KUKA KRL program: MyProgram_235().src

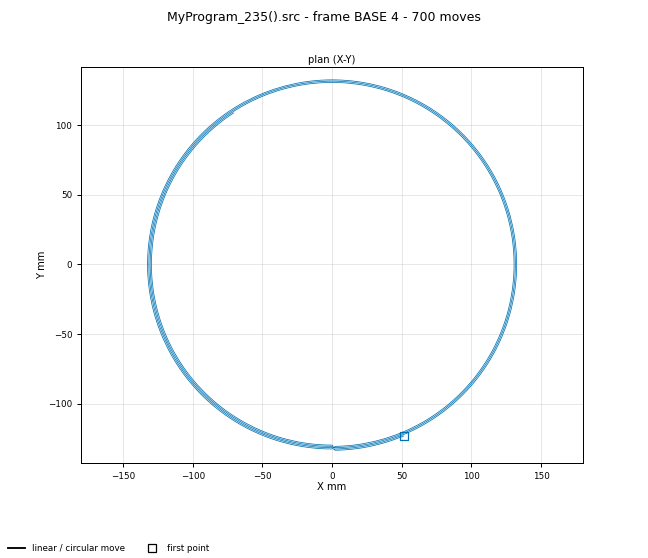
[picture p0: tool path of MyProgram_235().src in frame BASE 4, 700 of 700 moves have a stored position in this frame; points joined in program order, loops and branches not executed]
&ACCESS RVP
&REL 1
&PARAM TEMPLATE = C:\KRC\Roboter\Template\vorgabe
&PARAM EDITMASK = *
DEF MyProgram_235()
; ---- Setting reference (Base) ----
$BASE = BASE_DATA[4]

; --------------------------
; ---- Setting tool (TCP) ----
$TOOL = TOOL_DATA[3]
; --------------------------

$VEL.CP = VEL_APROX_PRINT
Startdeposition()
$VEL.CP = VEL_PRINT
LIN {X 51.31,Y -123.078,Z 159,A -69.1463,B 20.1877,C -0.5171,E1 20.2552,E2 517.2278} C_DIS
LIN {X 48.8194,Y -124.0882,Z 159,A -70.4431,B 20.1878,C -0.5093,E1 20.2518,E2 518.5433} C_DIS
LIN {X 45.4149,Y -125.3733,Z 159,A -71.9054,B 20.1878,C -0.5117,E1 20.248,E2 519.9947} C_DIS
LIN {X 42.7947,Y -126.2935,Z 159,A -73.4065,B 20.1881,C -0.497,E1 20.2439,E2 521.5347} C_DIS
LIN {X 39.7378,Y -127.2887,Z 159,A -74.6325,B 20.188,C -0.5021,E1 20.2407,E2 522.7431} C_DIS
LIN {X 36.4684,Y -128.2628,Z 159,A -75.8559,B 20.1878,C -0.511,E1 20.2375,E2 523.9381} C_DIS
LIN {X 32.9588,Y -129.208,Z 159,A -77.479,B 20.1878,C -0.5068,E1 20.2331,E2 525.5701} C_DIS
LIN {X 29.9233,Y -129.9447,Z 159,A -78.8692,B 20.1879,C -0.5035,E1 20.2293,E2 526.9673} C_DIS
LIN {X 25.1569,Y -130.9509,Z 159,A -81.0499,B 20.1881,C -0.498,E1 20.2233,E2 529.1604} C_DIS
LIN {X 20.69,Y -131.7308,Z 159,A -82.9211,B 20.1881,C -0.4999,E1 20.2181,E2 531.0236} C_DIS
LIN {X 17.7382,Y -132.161,Z 159,A -84.2195,B 20.1881,C -0.4984,E1 20.2145,E2 532.325} C_DIS
LIN {X 14.1081,Y -132.5971,Z 159,A -85.8476,B 20.1881,C -0.4951,E1 20.21,E2 533.9611} C_DIS
LIN {X 9.8352,Y -132.9824,Z 159,A -87.5814,B 20.1881,C -0.499,E1 20.2052,E2 535.6827} C_DIS
LIN {X 6.2788,Y -133.1983,Z 159,A -89.2049,B 20.1881,C -0.4945,E1 20.2006,E2 537.3184} C_DIS
LIN {X 2.1393,Y -133.3285,Z 159,A -90.8711,B 20.1881,C -0.4988,E1 20.196,E2 538.9717} C_DIS
LIN {X 2.1393,Y -133.3285,Z 159,A -90.8711,B 20.1881,C -0.4988,E1 20.196,E2 538.9717} C_DIS
Enddeposition()
LIN {X 0.915,Y -132.4111,Z 159,A -90.6799,B 18.9878,C -0.3693,E1 18.993,E2 539.0606} C_DIS
Startdeposition()
$VEL.CP = VEL_PRINT
LIN {X 3.9489,Y -132.359,Z 159,A -89.0902,B 18.9875,C -0.3807,E1 18.9975,E2 537.4365} C_DIS
LIN {X 8.1067,Y -132.1692,Z 159,A -87.3119,B 18.9875,C -0.3804,E1 19.0025,E2 535.66} C_DIS
LIN {X 11.2426,Y -131.9395,Z 159,A -85.8993,B 18.9875,C -0.3831,E1 19.0064,E2 534.2402} C_DIS
LIN {X 15.547,Y -131.5017,Z 159,A -84.0509,B 18.9875,C -0.3831,E1 19.0115,E2 532.3935} C_DIS
LIN {X 18.8161,Y -131.0738,Z 159,A -82.5998,B 18.9875,C -0.3849,E1 19.0156,E2 530.9384} C_DIS
LIN {X 23.141,Y -130.3798,Z 159,A -80.3181,B 18.9871,C -0.402,E1 19.022,E2 528.6076} C_DIS
LIN {X 27.1338,Y -129.6097,Z 159,A -79.0268,B 18.9875,C -0.3843,E1 19.0254,E2 527.3728} C_DIS
LIN {X 29.78,Y -129.0256,Z 159,A -77.8051,B 18.9875,C -0.3874,E1 19.0287,E2 526.144} C_DIS
LIN {X 33.8587,Y -128.0156,Z 159,A -75.9883,B 18.9874,C -0.389,E1 19.0336,E2 524.3258} C_DIS
LIN {X 37.1501,Y -127.0992,Z 159,A -73.7766,B 18.9867,C -0.4207,E1 19.0398,E2 522.022} C_DIS
LIN {X 42.6388,Y -125.3669,Z 159,A -72.0801,B 18.9873,C -0.3908,E1 19.0441,E2 520.4216} C_DIS
LIN {X 46.6963,Y -123.9106,Z 159,A -70.1681,B 18.9873,C -0.3951,E1 19.0491,E2 518.502} C_DIS
LIN {X 50.0421,Y -122.5986,Z 159,A -68.6914,B 18.9873,C -0.394,E1 19.0529,E2 517.0333} C_DIS
LIN {X 52.8027,Y -121.4341,Z 159,A -67.3975,B 18.9873,C -0.3957,E1 19.0562,E2 515.7384} C_DIS
LIN {X 55.6063,Y -120.1758,Z 159,A -66.0096,B 18.9872,C -0.4,E1 19.0598,E2 514.3419} C_DIS
LIN {X 59.0942,Y -118.501,Z 159,A -64.0272,B 18.9868,C -0.4154,E1 19.0648,E2 512.3197} C_DIS
LIN {X 62.2036,Y -116.8996,Z 159,A -62.8732,B 18.9871,C -0.4029,E1 19.0676,E2 511.2084} C_DIS
LIN {X 65.5736,Y -115.0431,Z 159,A -61.1039,B 18.9869,C -0.41,E1 19.0719,E2 509.4243} C_DIS
LIN {X 70.2696,Y -112.2358,Z 159,A -58.4917,B 18.9866,C -0.4245,E1 19.0782,E2 506.779} C_DIS
LIN {X 73.2793,Y -110.2952,Z 159,A -57.3437,B 18.9869,C -0.4106,E1 19.0808,E2 505.6786} C_DIS
LIN {X 76.3906,Y -108.1633,Z 159,A -55.3096,B 18.9865,C -0.4306,E1 19.0855,E2 503.5928} C_DIS
LIN {X 79.3344,Y -106.0234,Z 159,A -54.2415,B 18.9869,C -0.4125,E1 19.0878,E2 502.5853} C_DIS
LIN {X 82.0871,Y -103.9069,Z 159,A -52.6363,B 18.9867,C -0.4199,E1 19.0914,E2 500.9656} C_DIS
LIN {X 84.9344,Y -101.5923,Z 159,A -50.4502,B 18.9861,C -0.4485,E1 19.0962,E2 498.7032} C_DIS
LIN {X 88.5384,Y -98.4673,Z 159,A -48.5996,B 18.9862,C -0.4441,E1 19.1,E2 496.8764} C_DIS
LIN {X 91.2721,Y -95.9391,Z 159,A -47.5951,B 18.9867,C -0.4221,E1 19.1019,E2 495.9445} C_DIS
LIN {X 94.6689,Y -92.5885,Z 159,A -44.8289,B 18.9859,C -0.4566,E1 19.1076,E2 493.0888} C_DIS
LIN {X 97.6523,Y -89.4365,Z 159,A -42.7552,B 18.9856,C -0.4695,E1 19.1115,E2 490.988} C_DIS
LIN {X 101.2378,Y -85.357,Z 159,A -41.1575,B 18.9862,C -0.4433,E1 19.1142,E2 489.4802} C_DIS
LIN {X 104.3228,Y -81.557,Z 159,A -38.8266,B 18.9859,C -0.4578,E1 19.1183,E2 487.1199} C_DIS
LIN {X 106.4737,Y -78.7289,Z 159,A -36.881,B 18.9854,C -0.4792,E1 19.1217,E2 485.1214} C_DIS
LIN {X 109.3425,Y -74.6934,Z 159,A -35.5347,B 18.9861,C -0.451,E1 19.1237,E2 483.8704} C_DIS
LIN {X 111.0638,Y -72.1085,Z 159,A -33.9343,B 18.9857,C -0.4655,E1 19.1262,E2 482.2364} C_DIS
LIN {X 113.1829,Y -68.735,Z 159,A -32.2214,B 18.9857,C -0.4698,E1 19.1287,E2 480.5223} C_DIS
LIN {X 115.4009,Y -64.9419,Z 159,A -30.372,B 18.9855,C -0.4729,E1 19.1312,E2 478.6764} C_DIS
LIN {X 117.3378,Y -61.369,Z 159,A -28.6996,B 18.9855,C -0.4742,E1 19.1334,E2 477.0117} C_DIS
LIN {X 119.1222,Y -57.8349,Z 159,A -27.0067,B 18.9855,C -0.4783,E1 19.1355,E2 475.3187} C_DIS
LIN {X 120.4094,Y -55.1012,Z 159,A -25.6347,B 18.9852,C -0.4848,E1 19.1371,E2 473.9368} C_DIS
LIN {X 121.9652,Y -51.5668,Z 159,A -24.0045,B 18.9852,C -0.488,E1 19.1389,E2 472.309} C_DIS
LIN {X 124.4421,Y -45.2616,Z 159,A -21.3203,B 18.9852,C -0.4861,E1 19.1416,E2 469.6506} C_DIS
LIN {X 125.713,Y -41.6006,Z 159,A -19.4119,B 18.9848,C -0.5011,E1 19.1434,E2 467.7112} C_DIS
LIN {X 127.6951,Y -35.0529,Z 159,A -16.5806,B 18.9848,C -0.5045,E1 19.1456,E2 464.8912} C_DIS
LIN {X 128.3642,Y -32.5112,Z 159,A -15.4138,B 18.9846,C -0.5093,E1 19.1464,E2 463.7189} C_DIS
LIN {X 129.7937,Y -26.2296,Z 159,A -12.6235,B 18.9844,C -0.518,E1 19.1481,E2 460.924} C_DIS
LIN {X 130.7421,Y -21.0106,Z 159,A -10.3225,B 18.9842,C -0.5254,E1 19.1492,E2 458.6189} C_DIS
LIN {X 131.2848,Y -17.2825,Z 159,A -8.7108,B 18.9841,C -0.5297,E1 19.1498,E2 457.0068} C_DIS
LIN {X 131.7831,Y -12.9506,Z 159,A -6.9501,B 18.9841,C -0.5302,E1 19.1503,E2 455.2588} C_DIS
LIN {X 132.0586,Y -9.744,Z 159,A -5.47,B 18.9839,C -0.5383,E1 19.1507,E2 453.7658} C_DIS
LIN {X 132.2857,Y -5.9509,Z 159,A -3.646,B 18.9835,C -0.5511,E1 19.1509,E2 451.9174} C_DIS
LIN {X 132.4155,Y -0.8768,Z 159,A -1.6644,B 18.9835,C -0.5488,E1 19.151,E2 449.9587} C_DIS
LIN {X 132.3754,Y 3.3608,Z 159,A 0.1535,B 18.9835,C -0.5538,E1 19.151,E2 448.1401} C_DIS
LIN {X 132.2469,Y 6.7219,Z 159,A 1.588,B 18.9833,C -0.5575,E1 19.1507,E2 446.7061} C_DIS
LIN {X 132.0141,Y 10.3543,Z 159,A 3.2561,B 18.9831,C -0.5663,E1 19.1504,E2 445.0244} C_DIS
LIN {X 131.6494,Y 14.2426,Z 159,A 4.8067,B 18.9831,C -0.5656,E1 19.15,E2 443.4883} C_DIS
LIN {X 131.1522,Y 18.2677,Z 159,A 6.661,B 18.9828,C -0.5753,E1 19.1493,E2 441.6194} C_DIS
LIN {X 130.5569,Y 22.1221,Z 159,A 8.2165,B 18.9828,C -0.5748,E1 19.1486,E2 440.0777} C_DIS
LIN {X 129.5781,Y 27.2807,Z 159,A 11.5557,B 18.9812,C -0.6276,E1 19.1466,E2 436.6038} C_DIS
LIN {X 127.8681,Y 34.412,Z 159,A 13.1779,B 18.983,C -0.5706,E1 19.1457,E2 435.168} C_DIS
LIN {X 125.8783,Y 41.1045,Z 159,A 16.7762,B 18.982,C -0.6038,E1 19.1427,E2 431.496} C_DIS
LIN {X 124.582,Y 44.8736,Z 159,A 18.3588,B 18.982,C -0.6028,E1 19.1412,E2 429.9286} C_DIS
LIN {X 123.3427,Y 48.1759,Z 159,A 19.8352,B 18.982,C -0.6051,E1 19.1397,E2 428.4564} C_DIS
LIN {X 122.1018,Y 51.2397,Z 159,A 21.2099,B 18.9819,C -0.6068,E1 19.1383,E2 427.0868} C_DIS
LIN {X 120.8903,Y 54.0353,Z 159,A 22.5822,B 18.9817,C -0.6127,E1 19.1367,E2 425.7064} C_DIS
LIN {X 119.4225,Y 57.2063,Z 159,A 24.123,B 18.9815,C -0.6181,E1 19.1349,E2 424.1604} C_DIS
LIN {X 117.8596,Y 60.3613,Z 159,A 25.6041,B 18.9815,C -0.6205,E1 19.133,E2 422.6828} C_DIS
LIN {X 115.9936,Y 63.8779,Z 159,A 27.3655,B 18.9812,C -0.6267,E1 19.1307,E2 420.9149} C_DIS
LIN {X 113.9778,Y 67.4093,Z 159,A 29.1303,B 18.9811,C -0.6315,E1 19.1282,E2 419.1476} C_DIS
LIN {X 111.7699,Y 71.0102,Z 159,A 30.9547,B 18.9809,C -0.6361,E1 19.1255,E2 417.3219} C_DIS
LIN {X 109.3756,Y 74.6451,Z 159,A 32.839,B 18.9808,C -0.6409,E1 19.1226,E2 415.4356} C_DIS
LIN {X 106.7983,Y 78.2876,Z 159,A 34.7322,B 18.9807,C -0.644,E1 19.1195,E2 413.5452} C_DIS
LIN {X 104.0816,Y 81.8647,Z 159,A 36.6347,B 18.9806,C -0.6469,E1 19.1162,E2 411.6459} C_DIS
LIN {X 101.2742,Y 85.3136,Z 159,A 38.5288,B 18.9805,C -0.6501,E1 19.1129,E2 409.7539} C_DIS
LIN {X 98.4189,Y 88.5925,Z 159,A 40.6781,B 18.98,C -0.6655,E1 19.1088,E2 407.5706} C_DIS
LIN {X 96.1324,Y 91.0683,Z 159,A 41.8429,B 18.9803,C -0.6565,E1 19.1066,E2 406.4404} C_DIS
LIN {X 93.2493,Y 94.018,Z 159,A 43.6666,B 18.9801,C -0.6618,E1 19.103,E2 404.6107} C_DIS
LIN {X 90.0676,Y 97.0705,Z 159,A 45.5495,B 18.9801,C -0.6647,E1 19.0992,E2 402.7295} C_DIS
LIN {X 86.7928,Y 100.0097,Z 159,A 47.4911,B 18.9798,C -0.67,E1 19.0951,E2 400.7823} C_DIS
LIN {X 83.3209,Y 102.9199,Z 159,A 49.7722,B 18.9792,C -0.6869,E1 19.0901,E2 398.4612} C_DIS
LIN {X 80.1132,Y 105.4365,Z 159,A 50.9917,B 18.9799,C -0.6676,E1 19.0876,E2 397.3067} C_DIS
LIN {X 77.3722,Y 107.4641,Z 159,A 52.6714,B 18.9795,C -0.6785,E1 19.0837,E2 395.6017} C_DIS
LIN {X 73.6546,Y 110.0446,Z 159,A 54.5931,B 18.9795,C -0.6803,E1 19.0793,E2 393.6835} C_DIS
LIN {X 69.8977,Y 112.4683,Z 159,A 56.56,B 18.9793,C -0.6846,E1 19.0746,E2 391.7119} C_DIS
LIN {X 67.0765,Y 114.1734,Z 159,A 57.9282,B 18.9793,C -0.6843,E1 19.0714,E2 390.3503} C_DIS
LIN {X 63.0971,Y 116.4203,Z 159,A 59.8897,B 18.9793,C -0.6864,E1 19.0666,E2 388.3902} C_DIS
LIN {X 59.9293,Y 118.0796,Z 159,A 61.3421,B 18.9793,C -0.6846,E1 19.063,E2 386.9486} C_DIS
LIN {X 56.981,Y 119.5302,Z 159,A 62.779,B 18.9793,C -0.687,E1 19.0594,E2 385.5097} C_DIS
LIN {X 53.9235,Y 120.9404,Z 159,A 64.2047,B 18.9793,C -0.6874,E1 19.0558,E2 384.0874} C_DIS
LIN {X 51.0132,Y 122.1964,Z 159,A 65.602,B 18.9791,C -0.6899,E1 19.0522,E2 382.687} C_DIS
LIN {X 47.9779,Y 123.4197,Z 159,A 67.0215,B 18.9791,C -0.6915,E1 19.0485,E2 381.2669} C_DIS
LIN {X 44.6483,Y 124.6632,Z 159,A 68.4959,B 18.9791,C -0.6904,E1 19.0446,E2 379.8} C_DIS
LIN {X 41.5878,Y 125.7173,Z 159,A 69.9214,B 18.9791,C -0.6926,E1 19.0408,E2 378.3716} C_DIS
LIN {X 38.1357,Y 126.8086,Z 159,A 72.0247,B 18.9782,C -0.7153,E1 19.0351,E2 376.2037} C_DIS
LIN {X 33.9426,Y 127.9932,Z 159,A 72.9798,B 18.9795,C -0.6796,E1 19.0328,E2 375.3603} C_DIS
LIN {X 28.5936,Y 129.2947,Z 159,A 75.8626,B 18.9788,C -0.7007,E1 19.0248,E2 372.4183} C_DIS
LIN {X 25.4061,Y 129.9585,Z 159,A 77.2631,B 18.9788,C -0.7011,E1 19.021,E2 371.019} C_DIS
LIN {X 21.6945,Y 130.6282,Z 159,A 78.788,B 18.9788,C -0.6975,E1 19.0168,E2 369.5073} C_DIS
LIN {X 18.2684,Y 131.1521,Z 159,A 80.4878,B 18.9786,C -0.7058,E1 19.012,E2 367.784} C_DIS
LIN {X 14.5763,Y 131.6134,Z 159,A 81.9505,B 18.9788,C -0.7004,E1 19.008,E2 366.3394} C_DIS
LIN {X 11.0145,Y 131.9587,Z 159,A 83.472,B 18.9788,C -0.6996,E1 19.0038,E2 364.8217} C_DIS
LIN {X 6.8228,Y 132.2418,Z 159,A 85.2635,B 18.9788,C -0.6986,E1 18.9988,E2 363.034} C_DIS
LIN {X 3.5533,Y 132.37,Z 159,A 86.6449,B 18.9788,C -0.6973,E1 18.995,E2 361.6573} C_DIS
LIN {X -0.1185,Y 132.4191,Z 159,A 88.3711,B 18.9787,C -0.7024,E1 18.9901,E2 359.9156} C_DIS
LIN {X -4.1755,Y 132.3527,Z 159,A 90.021,B 18.9789,C -0.6979,E1 18.9855,E2 358.2792} C_DIS
LIN {X -7.9769,Y 132.1772,Z 159,A 91.6914,B 18.9789,C -0.6984,E1 18.9809,E2 356.6069} C_DIS
LIN {X -11.6377,Y 131.9061,Z 159,A 93.3916,B 18.9787,C -0.7021,E1 18.9761,E2 354.8943} C_DIS
LIN {X -16.3558,Y 131.4052,Z 159,A 95.2652,B 18.979,C -0.6941,E1 18.971,E2 353.0434} C_DIS
LIN {X -21.2273,Y 130.7062,Z 159,A 97.9516,B 18.9783,C -0.7143,E1 18.9634,E2 350.292} C_DIS
LIN {X -25.4199,Y 129.9558,Z 159,A 99.3428,B 18.9789,C -0.6956,E1 18.9597,E2 348.9562} C_DIS
LIN {X -33.9519,Y 127.9908,Z 159,A 102.871,B 18.9794,C -0.6824,E1 18.9503,E2 345.4622} C_DIS
LIN {X -41.8666,Y 125.6245,Z 159,A 106.3434,B 18.9797,C -0.6748,E1 18.941,E2 342.0054} C_DIS
LIN {X -45.3648,Y 124.4049,Z 159,A 108.2563,B 18.9793,C -0.6846,E1 18.9359,E2 340.0574} C_DIS
LIN {X -48.2073,Y 123.3305,Z 159,A 109.6279,B 18.9793,C -0.6851,E1 18.9323,E2 338.6803} C_DIS
LIN {X -55.1818,Y 120.3721,Z 159,A 112.7433,B 18.9797,C -0.6745,E1 18.9244,E2 335.5878} C_DIS
LIN {X -63.1056,Y 116.4157,Z 159,A 116.7481,B 18.9797,C -0.6749,E1 18.9143,E2 331.567} C_DIS
LIN {X -66.5151,Y 114.5015,Z 159,A 118.5527,B 18.9797,C -0.6763,E1 18.9099,E2 329.751} C_DIS
LIN {X -70.3547,Y 112.1836,Z 159,A 120.4927,B 18.9797,C -0.6729,E1 18.9053,E2 327.8134} C_DIS
LIN {X -73.8825,Y 109.8924,Z 159,A 122.3636,B 18.9797,C -0.6714,E1 18.9009,E2 325.9387} C_DIS
LIN {X -77.5373,Y 107.3443,Z 159,A 124.2871,B 18.9799,C -0.6676,E1 18.8966,E2 324.0181} C_DIS
LIN {X -81.3022,Y 104.5218,Z 159,A 126.2701,B 18.9801,C -0.6615,E1 18.8922,E2 322.044} C_DIS
LIN {X -84.6828,Y 101.8024,Z 159,A 128.177,B 18.9802,C -0.6587,E1 18.8881,E2 320.1361} C_DIS
LIN {X -87.9054,Y 99.0329,Z 159,A 130.0707,B 18.9802,C -0.6568,E1 18.8841,E2 318.2382} C_DIS
LIN {X -90.7085,Y 96.471,Z 159,A 132.1399,B 18.9799,C -0.6688,E1 18.8798,E2 316.1204} C_DIS
LIN {X -93.9041,Y 93.3639,Z 159,A 133.4787,B 18.9807,C -0.6427,E1 18.8773,E2 314.8547} C_DIS
LIN {X -96.5447,Y 90.6313,Z 159,A 135.3109,B 18.9807,C -0.6457,E1 18.8737,E2 313.0024} C_DIS
LIN {X -98.8382,Y 88.1244,Z 159,A 136.77,B 18.9807,C -0.6417,E1 18.871,E2 311.5468} C_DIS
LIN {X -101.7121,Y 84.7917,Z 159,A 138.7035,B 18.9809,C -0.6381,E1 18.8675,E2 309.6125} C_DIS
LIN {X -104.4223,Y 81.4306,Z 159,A 140.6191,B 18.9809,C -0.6351,E1 18.8642,E2 307.6941} C_DIS
LIN {X -107.1288,Y 77.8347,Z 159,A 142.5465,B 18.9812,C -0.6293,E1 18.861,E2 305.7719} C_DIS
LIN {X -109.7841,Y 74.0426,Z 159,A 144.56,B 18.9813,C -0.6244,E1 18.8578,E2 303.7601} C_DIS
LIN {X -112.2021,Y 70.3255,Z 159,A 146.4781,B 18.9815,C -0.6192,E1 18.8549,E2 301.845} C_DIS
LIN {X -114.3948,Y 66.6993,Z 159,A 148.3771,B 18.9815,C -0.6165,E1 18.8522,E2 299.941} C_DIS
LIN {X -117.4487,Y 61.1579,Z 159,A 151.0125,B 18.9819,C -0.6051,E1 18.8487,E2 297.3219} C_DIS
LIN {X -119.3241,Y 57.4124,Z 159,A 152.6406,B 18.9823,C -0.5933,E1 18.8467,E2 295.7185} C_DIS
LIN {X -120.3866,Y 55.1504,Z 159,A 153.9121,B 18.9822,C -0.597,E1 18.8452,E2 294.4261} C_DIS
LIN {X -121.7642,Y 52.0393,Z 159,A 155.4594,B 18.9822,C -0.5954,E1 18.8435,E2 292.8721} C_DIS
LIN {X -122.9857,Y 49.0818,Z 159,A 156.7759,B 18.9824,C -0.5889,E1 18.8421,E2 291.5659} C_DIS
LIN {X -124.0965,Y 46.2,Z 159,A 158.1239,B 18.9825,C -0.5853,E1 18.8408,E2 290.2185} C_DIS
LIN {X -125.134,Y 43.3106,Z 159,A 159.4706,B 18.9826,C -0.582,E1 18.8395,E2 288.8717} C_DIS
LIN {X -126.1487,Y 40.2595,Z 159,A 160.9216,B 18.9826,C -0.58,E1 18.8383,E2 287.4158} C_DIS
LIN {X -127.3031,Y 36.4538,Z 159,A 162.7606,B 18.9827,C -0.579,E1 18.8368,E2 285.5655} C_DIS
LIN {X -128.3116,Y 32.7185,Z 159,A 164.3503,B 18.9829,C -0.5708,E1 18.8357,E2 283.9884} C_DIS
LIN {X -129.2525,Y 28.7867,Z 159,A 166.2563,B 18.9829,C -0.5711,E1 18.8345,E2 282.0665} C_DIS
LIN {X -130.0542,Y 24.9051,Z 159,A 168.5833,B 18.9824,C -0.5879,E1 18.8333,E2 279.6686} C_DIS
LIN {X -131.0123,Y 19.2464,Z 159,A 170.1827,B 18.9836,C -0.5483,E1 18.8326,E2 278.179} C_DIS
LIN {X -131.7196,Y 13.5901,Z 159,A 172.8602,B 18.9836,C -0.5482,E1 18.8317,E2 275.4802} C_DIS
LIN {X -132.0376,Y 10.0315,Z 159,A 174.4321,B 18.9836,C -0.5443,E1 18.8314,E2 273.9075} C_DIS
LIN {X -132.2591,Y 6.479,Z 159,A 175.9477,B 18.9839,C -0.5386,E1 18.8311,E2 272.3971} C_DIS
LIN {X -132.4177,Y 0.4728,Z 159,A 178.8183,B 18.9839,C -0.5402,E1 18.8311,E2 269.498} C_DIS
LIN {X -132.3284,Y -4.8688,Z 159,A -179.0942,B 18.9842,C -0.5249,E1 18.8311,E2 267.4408} C_DIS
LIN {X -132.1346,Y -8.6683,Z 159,A -176.9755,B 18.9839,C -0.5369,E1 18.8316,E2 265.2678} C_DIS
LIN {X -131.7925,Y -12.8521,Z 159,A -175.7471,B 18.9846,C -0.5101,E1 18.8319,E2 264.1124} C_DIS
LIN {X -131.0279,Y -19.1375,Z 159,A -172.8894,B 18.9847,C -0.5058,E1 18.8329,E2 261.2446} C_DIS
LIN {X -130.2956,Y -23.6116,Z 159,A -170.025,B 18.984,C -0.5327,E1 18.8343,E2 258.274} C_DIS
LIN {X -129.0506,Y -29.6704,Z 159,A -168.1285,B 18.985,C -0.4962,E1 18.8354,E2 256.4754} C_DIS
LIN {X -128.0154,Y -33.8595,Z 159,A -166.3014,B 18.9851,C -0.4892,E1 18.8367,E2 254.6556} C_DIS
LIN {X -127.0089,Y -37.4586,Z 159,A -164.6666,B 18.9852,C -0.4851,E1 18.8379,E2 253.0207} C_DIS
LIN {X -126.074,Y -40.4935,Z 159,A -163.3365,B 18.9854,C -0.4794,E1 18.839,E2 251.6976} C_DIS
LIN {X -125.0422,Y -43.5753,Z 159,A -161.8377,B 18.9854,C -0.4787,E1 18.8404,E2 250.1894} C_DIS
LIN {X -122.7613,Y -49.6387,Z 159,A -159.0527,B 18.9856,C -0.4701,E1 18.8432,E2 247.4101} C_DIS
LIN {X -121.2331,Y -53.2676,Z 159,A -156.5303,B 18.985,C -0.4953,E1 18.8461,E2 244.7907} C_DIS
LIN {X -118.7944,Y -58.4995,Z 159,A -155.1214,B 18.9861,C -0.4486,E1 18.8477,E2 243.5161} C_DIS
LIN {X -117.8133,Y -60.4523,Z 159,A -153.8318,B 18.9859,C -0.4585,E1 18.8493,E2 242.1863} C_DIS
LIN {X -115.7052,Y -64.3987,Z 159,A -151.6623,B 18.9858,C -0.4619,E1 18.8523,E2 239.9907} C_DIS
LIN {X -113.1193,Y -68.8402,Z 159,A -149.5644,B 18.986,C -0.4515,E1 18.8553,E2 237.9103} C_DIS
LIN {X -109.3146,Y -74.734,Z 159,A -146.865,B 18.9865,C -0.4315,E1 18.8593,E2 235.2544} C_DIS
LIN {X -106.4425,Y -78.7715,Z 159,A -144.3369,B 18.9863,C -0.4404,E1 18.8635,E2 232.682} C_DIS
LIN {X -102.7434,Y -83.5386,Z 159,A -142.0415,B 18.9867,C -0.4226,E1 18.8674,E2 230.427} C_DIS
LIN {X -98.1856,Y -88.8505,Z 159,A -138.7986,B 18.9867,C -0.4237,E1 18.8734,E2 227.1608} C_DIS
LIN {X -95.4574,Y -91.7761,Z 159,A -136.9399,B 18.9867,C -0.4248,E1 18.877,E2 225.2878} C_DIS
LIN {X -92.3875,Y -94.8657,Z 159,A -134.7656,B 18.9865,C -0.4318,E1 18.8814,E2 223.0797} C_DIS
LIN {X -89.719,Y -97.3926,Z 159,A -133.5799,B 18.9869,C -0.4134,E1 18.8837,E2 221.9441} C_DIS
LIN {X -86.7673,Y -100.032,Z 159,A -131.1902,B 18.9864,C -0.4356,E1 18.8889,E2 219.4732} C_DIS
LIN {X -82.9238,Y -103.2401,Z 159,A -129.6745,B 18.987,C -0.4071,E1 18.892,E2 218.0379} C_DIS
LIN {X -80.0418,Y -105.4904,Z 159,A -127.9361,B 18.987,C -0.4102,E1 18.8959,E2 216.2814} C_DIS
LIN {X -76.3541,Y -108.189,Z 159,A -126.0358,B 18.987,C -0.4039,E1 18.9002,E2 214.3913} C_DIS
LIN {X -72.9711,Y -110.4991,Z 159,A -124.1954,B 18.987,C -0.4037,E1 18.9045,E2 212.5435} C_DIS
LIN {X -69.1342,Y -112.9393,Z 159,A -122.0649,B 18.987,C -0.407,E1 18.9096,E2 210.3937} C_DIS
LIN {X -65.223,Y -115.2429,Z 159,A -120.2149,B 18.9872,C -0.3998,E1 18.914,E2 208.5584} C_DIS
LIN {X -61.6467,Y -117.192,Z 159,A -118.5871,B 18.9873,C -0.3924,E1 18.918,E2 206.9472} C_DIS
LIN {X -58.303,Y -118.8913,Z 159,A -116.9679,B 18.9873,C -0.3903,E1 18.922,E2 205.3289} C_DIS
LIN {X -55.3221,Y -120.3072,Z 159,A -115.5388,B 18.9873,C -0.3887,E1 18.9256,E2 203.8999} C_DIS
LIN {X -52.3693,Y -121.6215,Z 159,A -114.1327,B 18.9874,C -0.3874,E1 18.9292,E2 202.493} C_DIS
LIN {X -49.1351,Y -122.9642,Z 159,A -112.6136,B 18.9874,C -0.3861,E1 18.9332,E2 200.9737} C_DIS
LIN {X -46.2,Y -124.0965,Z 159,A -111.2497,B 18.9874,C -0.3849,E1 18.9367,E2 199.6095} C_DIS
LIN {X -42.7901,Y -125.3144,Z 159,A -109.6999,B 18.9874,C -0.3829,E1 18.9408,E2 198.0619} C_DIS
LIN {X -37.4635,Y -127.0074,Z 159,A -107.3061,B 18.9875,C -0.3801,E1 18.9472,E2 195.671} C_DIS
LIN {X -30.1193,Y -128.9481,Z 159,A -104.0276,B 18.9875,C -0.3777,E1 18.9561,E2 192.3934} C_DIS
LIN {X -26.0153,Y -129.8373,Z 159,A -102.0249,B 18.9875,C -0.3841,E1 18.9616,E2 190.3676} C_DIS
LIN {X -21.725,Y -130.6231,Z 159,A -100.2544,B 18.9875,C -0.3789,E1 18.9664,E2 188.611} C_DIS
LIN {X -18.6904,Y -131.0918,Z 159,A -98.9167,B 18.9875,C -0.3789,E1 18.9701,E2 187.2719} C_DIS
LIN {X -14.9487,Y -131.5731,Z 159,A -97.1696,B 18.9875,C -0.3831,E1 18.975,E2 185.5102} C_DIS
LIN {X -11.1625,Y -131.9462,Z 159,A -95.6353,B 18.9875,C -0.3785,E1 18.9792,E2 183.9889} C_DIS
LIN {X -7.8986,Y -132.182,Z 159,A -94.2493,B 18.9876,C -0.3773,E1 18.9831,E2 182.6061} C_DIS
LIN {X -4.108,Y -132.3546,Z 159,A -92.511,B 18.9876,C -0.3812,E1 18.988,E2 180.8553} C_DIS
LIN {X -0.1031,Y -132.4191,Z 159,A -90.7238,B 18.9875,C -0.3836,E1 18.993,E2 179.0606} C_DIS
LIN {X -0.1031,Y -132.4191,Z 159,A -90.7238,B 18.9875,C -0.3836,E1 18.993,E2 179.0606} C_DIS
Enddeposition()
LIN {X 0.9129,Y -131.485,Z 159,A -90.5239,B 17.4908,C -0.1959,E1 17.4928,E2 179.345} C_DIS
Startdeposition()
$VEL.CP = VEL_PRINT
LIN {X -2.2876,Y -131.4698,Z 159,A -92.0327,B 17.4908,C -0.1916,E1 17.4886,E2 180.8682} C_DIS
LIN {X -6.4242,Y -131.3327,Z 159,A -93.8109,B 17.4908,C -0.1924,E1 17.4836,E2 182.6441} C_DIS
LIN {X -9.9377,Y -131.114,Z 159,A -95.3295,B 17.4908,C -0.193,E1 17.4794,E2 184.1616} C_DIS
LIN {X -13.5576,Y -130.7898,Z 159,A -96.9962,B 17.4909,C -0.1903,E1 17.4747,E2 185.8388} C_DIS
LIN {X -17.1749,Y -130.363,Z 159,A -98.5027,B 17.4909,C -0.1935,E1 17.4706,E2 187.336} C_DIS
LIN {X -20.1643,Y -129.9342,Z 159,A -99.8208,B 17.4909,C -0.1938,E1 17.4669,E2 188.6548} C_DIS
LIN {X -23.5365,Y -129.3663,Z 159,A -101.2915,B 17.4909,C -0.195,E1 17.4629,E2 190.1235} C_DIS
LIN {X -27.242,Y -128.6375,Z 159,A -103.0672,B 17.4909,C -0.1911,E1 17.458,E2 191.9152} C_DIS
LIN {X -33.831,Y -127.0626,Z 159,A -105.6197,B 17.4907,C -0.2069,E1 17.4512,E2 194.4204} C_DIS
LIN {X -40.438,Y -125.1175,Z 159,A -108.888,B 17.4908,C -0.1996,E1 17.4424,E2 197.721} C_DIS
LIN {X -43.3103,Y -124.1519,Z 159,A -110.2523,B 17.4908,C -0.1992,E1 17.4387,E2 199.0905} C_DIS
LIN {X -46.3411,Y -123.0527,Z 159,A -111.6572,B 17.4908,C -0.2004,E1 17.4351,E2 200.4954} C_DIS
LIN {X -49.3774,Y -121.866,Z 159,A -113.0621,B 17.4908,C -0.2024,E1 17.4314,E2 201.8983} C_DIS
LIN {X -52.217,Y -120.6764,Z 159,A -114.4659,B 17.4908,C -0.2016,E1 17.4278,E2 203.3094} C_DIS
LIN {X -55.5315,Y -119.188,Z 159,A -116.0286,B 17.4908,C -0.2041,E1 17.4238,E2 204.8695} C_DIS
LIN {X -58.5664,Y -117.7266,Z 159,A -117.4978,B 17.4908,C -0.2058,E1 17.4201,E2 206.3386} C_DIS
LIN {X -62.063,Y -115.9229,Z 159,A -119.2572,B 17.4908,C -0.2065,E1 17.4158,E2 208.1031} C_DIS
LIN {X -65.5102,Y -114.0109,Z 159,A -121.0811,B 17.4908,C -0.2052,E1 17.4113,E2 209.9391} C_DIS
LIN {X -69.8468,Y -111.4069,Z 159,A -123.0263,B 17.4906,C -0.2172,E1 17.4068,E2 211.853} C_DIS
LIN {X -72.6216,Y -109.6182,Z 159,A -124.7202,B 17.4906,C -0.2107,E1 17.4027,E2 213.5767} C_DIS
LIN {X -76.1978,Y -107.1631,Z 159,A -126.6394,B 17.4906,C -0.2128,E1 17.3983,E2 215.4986} C_DIS
LIN {X -79.9092,Y -104.4243,Z 159,A -128.595,B 17.4906,C -0.2181,E1 17.394,E2 217.4468} C_DIS
LIN {X -85.5378,Y -99.8664,Z 159,A -131.8696,B 17.4906,C -0.2199,E1 17.3869,E2 220.7339} C_DIS
LIN {X -89.0171,Y -96.7774,Z 159,A -134.0909,B 17.4906,C -0.2174,E1 17.3823,E2 222.9769} C_DIS
LIN {X -91.5546,Y -94.3805,Z 159,A -135.092,B 17.4903,C -0.2378,E1 17.3804,E2 223.9157} C_DIS
LIN {X -93.6046,Y -92.3485,Z 159,A -136.6608,B 17.4904,C -0.23,E1 17.3772,E2 225.5205} C_DIS
LIN {X -96.6899,Y -89.1123,Z 159,A -139.2816,B 17.4907,C -0.212,E1 17.3721,E2 228.2187} C_DIS
LIN {X -100.4737,Y -84.824,Z 159,A -140.8298,B 17.4902,C -0.2486,E1 17.3695,E2 229.6545} C_DIS
LIN {X -103.7334,Y -80.8047,Z 159,A -143.0862,B 17.4902,C -0.2537,E1 17.3655,E2 231.9094} C_DIS
LIN {X -105.4592,Y -78.5383,Z 159,A -144.6195,B 17.4902,C -0.247,E1 17.3629,E2 233.4761} C_DIS
LIN {X -108.1461,Y -74.7961,Z 159,A -147.1892,B 17.4904,C -0.2335,E1 17.3587,E2 236.1099} C_DIS
LIN {X -110.8798,Y -70.6796,Z 159,A -148.7865,B 17.4901,C -0.257,E1 17.3563,E2 237.6402} C_DIS
LIN {X -112.8805,Y -67.4382,Z 159,A -150.6134,B 17.4901,C -0.2558,E1 17.3537,E2 239.4852} C_DIS
LIN {X -114.8175,Y -64.0858,Z 159,A -152.1686,B 17.49,C -0.2644,E1 17.3516,E2 241.0233} C_DIS
LIN {X -116.931,Y -60.1401,Z 159,A -154.1214,B 17.4899,C -0.2696,E1 17.349,E2 242.9744} C_DIS
LIN {X -120.9554,Y -51.5716,Z 159,A -158.1362,B 17.4897,C -0.2843,E1 17.3444,E2 246.9722} C_DIS
LIN {X -123.4358,Y -45.3167,Z 159,A -161.2183,B 17.4897,C -0.2877,E1 17.3412,E2 250.0687} C_DIS
LIN {X -124.6968,Y -41.7154,Z 159,A -162.8369,B 17.4895,C -0.2939,E1 17.3397,E2 251.6802} C_DIS
LIN {X -125.7032,Y -38.5765,Z 159,A -164.3099,B 17.4895,C -0.2968,E1 17.3385,E2 253.1558} C_DIS
LIN {X -126.6826,Y -35.2276,Z 159,A -165.8391,B 17.4894,C -0.301,E1 17.3373,E2 254.6842} C_DIS
LIN {X -127.6699,Y -31.469,Z 159,A -167.6613,B 17.4894,C -0.3018,E1 17.3361,E2 256.5195} C_DIS
LIN {X -129.3696,Y -23.5185,Z 159,A -171.1826,B 17.4892,C -0.3131,E1 17.3341,E2 260.0338} C_DIS
LIN {X -130.002,Y -19.7259,Z 159,A -173.6244,B 17.4895,C -0.2937,E1 17.3331,E2 262.5622} C_DIS
LIN {X -130.7484,Y -13.942,Z 159,A -174.9861,B 17.4887,C -0.3391,E1 17.3327,E2 263.7836} C_DIS
LIN {X -131.2595,Y -7.7823,Z 159,A -177.8756,B 17.4887,C -0.3409,E1 17.332,E2 266.6927} C_DIS
LIN {X -131.3911,Y -5.0914,Z 159,A -179.9134,B 17.4891,C -0.3169,E1 17.3317,E2 268.8292} C_DIS
LIN {X -131.4918,Y -0.0347,Z 159,A 177.75,B 17.4891,C -0.3195,E1 17.3317,E2 271.1781} C_DIS
LIN {X -131.3794,Y 5.3916,Z 159,A 176.1216,B 17.4885,C -0.3502,E1 17.3319,E2 272.718} C_DIS
LIN {X -131.1008,Y 10.1092,Z 159,A 174.0796,B 17.4884,C -0.3571,E1 17.3322,E2 274.7551} C_DIS
LIN {X -130.8645,Y 12.8082,Z 159,A 172.8386,B 17.4884,C -0.3588,E1 17.3326,E2 276.0015} C_DIS
LIN {X -130.4926,Y 16.1719,Z 159,A 171.255,B 17.4884,C -0.3598,E1 17.3331,E2 277.5957} C_DIS
LIN {X -129.9337,Y 20.1671,Z 159,A 169.1288,B 17.4884,C -0.3535,E1 17.334,E2 279.7619} C_DIS
LIN {X -129.2486,Y 24.1771,Z 159,A 167.923,B 17.488,C -0.3769,E1 17.3346,E2 280.8995} C_DIS
LIN {X -128.71,Y 26.9016,Z 159,A 166.3317,B 17.4881,C -0.3684,E1 17.3355,E2 282.5334} C_DIS
LIN {X -127.8088,Y 30.8927,Z 159,A 164.7966,B 17.4879,C -0.3818,E1 17.3364,E2 284.0371} C_DIS
LIN {X -127.0266,Y 33.9662,Z 159,A 163.3588,B 17.4879,C -0.3841,E1 17.3375,E2 285.4793} C_DIS
LIN {X -125.9696,Y 37.7056,Z 159,A 161.5224,B 17.4879,C -0.3846,E1 17.3389,E2 287.33} C_DIS
LIN {X -124.7095,Y 41.6771,Z 159,A 159.8377,B 17.4876,C -0.3942,E1 17.3403,E2 288.9967} C_DIS
LIN {X -123.4561,Y 45.2603,Z 159,A 158.0673,B 17.4876,C -0.3953,E1 17.342,E2 290.7783} C_DIS
LIN {X -121.8224,Y 49.4858,Z 159,A 156.1955,B 17.4874,C -0.4044,E1 17.3439,E2 292.6352} C_DIS
LIN {X -120.5522,Y 52.5042,Z 159,A 154.7288,B 17.4874,C -0.4072,E1 17.3455,E2 294.1045} C_DIS
LIN {X -119.014,Y 55.9075,Z 159,A 153.107,B 17.4872,C -0.412,E1 17.3474,E2 295.7234} C_DIS
LIN {X -117.4188,Y 59.1818,Z 159,A 150.7221,B 17.4877,C -0.391,E1 17.3505,E2 298.1978} C_DIS
LIN {X -114.7498,Y 64.2064,Z 159,A 149.0988,B 17.4869,C -0.4252,E1 17.3526,E2 299.7191} C_DIS
LIN {X -113.1058,Y 67.0603,Z 159,A 147.4612,B 17.4869,C -0.4225,E1 17.3549,E2 301.378} C_DIS
LIN {X -110.8779,Y 70.6829,Z 159,A 145.57,B 17.4869,C -0.4263,E1 17.3577,E2 303.271} C_DIS
LIN {X -108.4326,Y 74.3794,Z 159,A 143.6487,B 17.4867,C -0.4317,E1 17.3607,E2 305.1884} C_DIS
LIN {X -105.9336,Y 77.8972,Z 159,A 141.7526,B 17.4867,C -0.436,E1 17.3638,E2 307.0837} C_DIS
LIN {X -103.1688,Y 81.5245,Z 159,A 139.7285,B 17.4865,C -0.4398,E1 17.3673,E2 309.1093} C_DIS
LIN {X -100.386,Y 84.9273,Z 159,A 137.8106,B 17.4865,C -0.4444,E1 17.3707,E2 311.0249} C_DIS
LIN {X -97.3432,Y 88.398,Z 159,A 135.8189,B 17.4863,C -0.4498,E1 17.3744,E2 313.0116} C_DIS
LIN {X -94.4278,Y 91.5057,Z 159,A 133.9286,B 17.4863,C -0.453,E1 17.378,E2 314.9033} C_DIS
LIN {X -89.1863,Y 96.6219,Z 159,A 130.9498,B 17.4859,C -0.4671,E1 17.384,E2 317.8533} C_DIS
LIN {X -86.7952,Y 98.7758,Z 159,A 129.2683,B 17.486,C -0.4609,E1 17.3875,E2 319.5654} C_DIS
LIN {X -83.4293,Y 101.6343,Z 159,A 127.327,B 17.486,C -0.4643,E1 17.3917,E2 321.5062} C_DIS
LIN {X -79.5589,Y 104.6922,Z 159,A 125.1705,B 17.4858,C -0.4683,E1 17.3964,E2 323.6609} C_DIS
LIN {X -75.9894,Y 107.3107,Z 159,A 123.2461,B 17.4858,C -0.4722,E1 17.4008,E2 325.5824} C_DIS
LIN {X -72.384,Y 109.7746,Z 159,A 121.3429,B 17.4856,C -0.4756,E1 17.4052,E2 327.4834} C_DIS
LIN {X -68.496,Y 112.2421,Z 159,A 119.3168,B 17.4856,C -0.4784,E1 17.41,E2 329.5096} C_DIS
LIN {X -64.7016,Y 114.4715,Z 159,A 117.3874,B 17.4855,C -0.4812,E1 17.4147,E2 331.4382} C_DIS
LIN {X -58.3681,Y 117.8245,Z 159,A 114.5575,B 17.4851,C -0.4958,E1 17.4216,E2 334.2308} C_DIS
LIN {X -55.5064,Y 119.1997,Z 159,A 112.187,B 17.4859,C -0.4648,E1 17.4279,E2 336.7136} C_DIS
LIN {X -50.3065,Y 121.4859,Z 159,A 110.5183,B 17.4851,C -0.495,E1 17.4319,E2 338.2873} C_DIS
LIN {X -47.3672,Y 122.6615,Z 159,A 109.0877,B 17.4851,C -0.495,E1 17.4356,E2 339.7225} C_DIS
LIN {X -43.4269,Y 124.1115,Z 159,A 107.1243,B 17.4851,C -0.4925,E1 17.4408,E2 341.6997} C_DIS
LIN {X -37.487,Y 126.0336,Z 159,A 104.6441,B 17.4849,C -0.5035,E1 17.4474,E2 344.1496} C_DIS
LIN {X -33.8503,Y 127.0575,Z 159,A 102.252,B 17.4855,C -0.4797,E1 17.454,E2 346.6265} C_DIS
LIN {X -29.0712,Y 128.2356,Z 159,A 100.6735,B 17.485,C -0.5007,E1 17.4581,E2 348.1381} C_DIS
LIN {X -20.9366,Y 129.8139,Z 159,A 97.158,B 17.4848,C -0.5064,E1 17.4678,E2 351.64} C_DIS
LIN {X -17.9952,Y 130.2537,Z 159,A 95.7706,B 17.4848,C -0.504,E1 17.4716,E2 353.0372} C_DIS
LIN {X -15.1794,Y 130.611,Z 159,A 94.447,B 17.4849,C -0.5016,E1 17.4753,E2 354.3701} C_DIS
LIN {X -11.0728,Y 131.0225,Z 159,A 92.7615,B 17.4849,C -0.5062,E1 17.4799,E2 356.0413} C_DIS
LIN {X -7.0275,Y 131.3024,Z 159,A 90.9256,B 17.4849,C -0.5044,E1 17.4851,E2 357.8843} C_DIS
LIN {X -2.9351,Y 131.4588,Z 159,A 89.0815,B 17.4849,C -0.5026,E1 17.4902,E2 359.7344} C_DIS
LIN {X 1.2172,Y 131.485,Z 159,A 87.2917,B 17.4849,C -0.5035,E1 17.4952,E2 361.521} C_DIS
LIN {X 5.1768,Y 131.3877,Z 159,A 85.6758,B 17.4848,C -0.5074,E1 17.4997,E2 363.1233} C_DIS
LIN {X 8.8014,Y 131.1967,Z 159,A 83.9757,B 17.4848,C -0.5031,E1 17.5045,E2 364.8367} C_DIS
LIN {X 12.7189,Y 130.8731,Z 159,A 82.4154,B 17.4848,C -0.5083,E1 17.5088,E2 366.3785} C_DIS
LIN {X 16.3574,Y 130.4697,Z 159,A 80.5966,B 17.485,C -0.5,E1 17.5139,E2 368.2229} C_DIS
LIN {X 20.1975,Y 129.929,Z 159,A 79.1007,B 17.4848,C -0.5063,E1 17.518,E2 369.6958} C_DIS
LIN {X 24.0279,Y 129.2772,Z 159,A 77.307,B 17.4849,C -0.502,E1 17.5229,E2 371.5008} C_DIS
LIN {X 27.4068,Y 128.6019,Z 159,A 75.7864,B 17.4849,C -0.5006,E1 17.5271,E2 373.0233} C_DIS
LIN {X 31.4996,Y 127.6626,Z 159,A 73.9638,B 17.4849,C -0.4997,E1 17.532,E2 374.8449} C_DIS
LIN {X 37.5306,Y 126.0209,Z 159,A 71.3929,B 17.4849,C -0.5032,E1 17.5389,E2 377.3977} C_DIS
LIN {X 40.6776,Y 125.041,Z 159,A 69.9681,B 17.4849,C -0.5025,E1 17.5427,E2 378.8212} C_DIS
LIN {X 43.3679,Y 124.132,Z 159,A 68.6974,B 17.4849,C -0.5002,E1 17.546,E2 380.0956} C_DIS
LIN {X 46.6066,Y 122.9533,Z 159,A 67.1308,B 17.4851,C -0.4964,E1 17.5502,E2 381.6699} C_DIS
LIN {X 50.4087,Y 121.4432,Z 159,A 65.3818,B 17.4851,C -0.4958,E1 17.5547,E2 383.415} C_DIS
LIN {X 53.5699,Y 120.082,Z 159,A 63.8868,B 17.4851,C -0.4943,E1 17.5585,E2 384.9097} C_DIS
LIN {X 56.9376,Y 118.5225,Z 159,A 62.3568,B 17.4851,C -0.4955,E1 17.5623,E2 386.4297} C_DIS
LIN {X 59.9324,Y 117.0367,Z 159,A 60.8502,B 17.4852,C -0.4918,E1 17.5661,E2 387.9424} C_DIS
LIN {X 63.5793,Y 115.0982,Z 159,A 58.9922,B 17.4853,C -0.4872,E1 17.5707,E2 389.8078} C_DIS
LIN {X 67.3884,Y 112.9102,Z 159,A 57.0269,B 17.4855,C -0.4826,E1 17.5754,E2 391.7796} C_DIS
LIN {X 71.3368,Y 110.4585,Z 159,A 55.0318,B 17.4855,C -0.4806,E1 17.5801,E2 393.7719} C_DIS
LIN {X 75.2518,Y 107.829,Z 159,A 53.0117,B 17.4855,C -0.4785,E1 17.5848,E2 395.7886} C_DIS
LIN {X 78.7838,Y 105.2764,Z 159,A 51.0651,B 17.4857,C -0.4734,E1 17.5892,E2 397.7416} C_DIS
LIN {X 83.7194,Y 101.3953,Z 159,A 48.5725,B 17.4856,C -0.4775,E1 17.5946,E2 400.2069} C_DIS
LIN {X 86.3835,Y 99.1353,Z 159,A 46.9033,B 17.4858,C -0.4691,E1 17.5981,E2 401.8943} C_DIS
LIN {X 89.6821,Y 96.1615,Z 159,A 44.9794,B 17.4858,C -0.4657,E1 17.6021,E2 403.8179} C_DIS
LIN {X 92.9264,Y 93.0307,Z 159,A 42.9903,B 17.486,C -0.4607,E1 17.6061,E2 405.8111} C_DIS
LIN {X 96.1308,Y 89.715,Z 159,A 40.8507,B 17.4863,C -0.4515,E1 17.6102,E2 407.9674} C_DIS
LIN {X 99.5539,Y 85.9007,Z 159,A 38.8039,B 17.4863,C -0.4536,E1 17.614,E2 409.9939} C_DIS
LIN {X 102.2018,Y 82.733,Z 159,A 37.0017,B 17.4863,C -0.4493,E1 17.6172,E2 411.7979} C_DIS
LIN {X 105.0266,Y 79.1159,Z 159,A 35.0715,B 17.4863,C -0.4472,E1 17.6204,E2 413.7214} C_DIS
LIN {X 107.6259,Y 75.5424,Z 159,A 33.1329,B 17.4865,C -0.4421,E1 17.6236,E2 415.6632} C_DIS
LIN {X 110.0812,Y 71.9179,Z 159,A 31.2447,B 17.4865,C -0.438,E1 17.6265,E2 417.5508} C_DIS
LIN {X 112.3289,Y 68.354,Z 159,A 29.3613,B 17.4867,C -0.4316,E1 17.6293,E2 419.4415} C_DIS
LIN {X 114.5994,Y 64.474,Z 159,A 27.5022,B 17.4867,C -0.4303,E1 17.6319,E2 421.2906} C_DIS
LIN {X 116.4136,Y 61.1332,Z 159,A 25.9043,B 17.4868,C -0.4281,E1 17.634,E2 422.8832} C_DIS
LIN {X 118.0364,Y 57.9384,Z 159,A 24.3135,B 17.487,C -0.4228,E1 17.636,E2 424.479} C_DIS
LIN {X 119.5363,Y 54.7784,Z 159,A 22.9148,B 17.487,C -0.4234,E1 17.6376,E2 425.8644} C_DIS
LIN {X 120.6751,Y 52.2198,Z 159,A 21.6294,B 17.487,C -0.4176,E1 17.639,E2 427.1588} C_DIS
LIN {X 121.9937,Y 49.0606,Z 159,A 20.1704,B 17.4871,C -0.4147,E1 17.6406,E2 428.6156} C_DIS
LIN {X 123.138,Y 46.1135,Z 159,A 18.7745,B 17.4872,C -0.4101,E1 17.642,E2 430.0152} C_DIS
LIN {X 124.3303,Y 42.7959,Z 159,A 17.2468,B 17.4873,C -0.406,E1 17.6434,E2 431.5437} C_DIS
LIN {X 126.3549,Y 36.3897,Z 159,A 14.4204,B 17.4874,C -0.4014,E1 17.6457,E2 434.3616} C_DIS
LIN {X 127.136,Y 33.5559,Z 159,A 12.869,B 17.4878,C -0.3872,E1 17.6469,E2 435.9466} C_DIS
LIN {X 128.4888,Y 27.9308,Z 159,A 10.0173,B 17.4882,C -0.367,E1 17.6487,E2 438.8406} C_DIS
LIN {X 129.4064,Y 23.3125,Z 159,A 8.5639,B 17.4878,C -0.3839,E1 17.6494,E2 440.2257} C_DIS
LIN {X 130.0144,Y 19.6464,Z 159,A 6.9776,B 17.4878,C -0.3802,E1 17.6501,E2 441.8102} C_DIS
LIN {X 130.5464,Y 15.7212,Z 159,A 5.2312,B 17.488,C -0.3742,E1 17.6507,E2 443.5613} C_DIS
LIN {X 130.9521,Y 11.896,Z 159,A 3.5231,B 17.4882,C -0.3678,E1 17.6511,E2 445.2755} C_DIS
LIN {X 131.24,Y 8.0991,Z 159,A 1.9756,B 17.4882,C -0.3671,E1 17.6514,E2 446.8119} C_DIS
LIN {X 131.4043,Y 4.7522,Z 159,A 0.4101,B 17.4883,C -0.3585,E1 17.6516,E2 448.3919} C_DIS
LIN {X 131.4891,Y 0.5912,Z 159,A -1.3175,B 17.4883,C -0.3563,E1 17.6516,E2 450.1117} C_DIS
LIN {X 131.4478,Y -3.3355,Z 159,A -3.0631,B 17.4885,C -0.3497,E1 17.6516,E2 451.8639} C_DIS
LIN {X 131.2862,Y -7.348,Z 159,A -4.8732,B 17.4887,C -0.3419,E1 17.6514,E2 453.6837} C_DIS
LIN {X 130.9958,Y -11.3895,Z 159,A -6.5068,B 17.4887,C -0.3416,E1 17.651,E2 455.304} C_DIS
LIN {X 130.5232,Y -15.9161,Z 159,A -8.4917,B 17.4887,C -0.3354,E1 17.6504,E2 457.292} C_DIS
LIN {X 129.9852,Y -19.8347,Z 159,A -10.7117,B 17.4892,C -0.3109,E1 17.6495,E2 459.5735} C_DIS
LIN {X 129.2123,Y -24.3672,Z 159,A -11.994,B 17.4888,C -0.3327,E1 17.6489,E2 460.7727} C_DIS
LIN {X 127.7509,Y -31.1329,Z 159,A -14.8868,B 17.4889,C -0.3283,E1 17.6472,E2 463.6553} C_DIS
LIN {X 125.9512,Y -37.7661,Z 159,A -18.0561,B 17.4892,C -0.3124,E1 17.6448,E2 466.8502} C_DIS
LIN {X 125.1412,Y -40.3638,Z 159,A -19.235,B 17.4892,C -0.3092,E1 17.6438,E2 468.03} C_DIS
LIN {X 124.2059,Y -43.1546,Z 159,A -20.5365,B 17.4893,C -0.3046,E1 17.6426,E2 469.3356} C_DIS
LIN {X 122.6362,Y -47.4308,Z 159,A -23.0799,B 17.4898,C -0.2772,E1 17.64,E2 471.9485} C_DIS
LIN {X 120.8619,Y -51.788,Z 159,A -24.3806,B 17.4894,C -0.3002,E1 17.6387,E2 473.1628} C_DIS
LIN {X 119.2685,Y -55.3576,Z 159,A -26.2751,B 17.4896,C -0.2879,E1 17.6365,E2 475.0827} C_DIS
LIN {X 117.8849,Y -58.2457,Z 159,A -27.6353,B 17.4896,C -0.2853,E1 17.6348,E2 476.4407} C_DIS
LIN {X 116.0265,Y -61.8703,Z 159,A -29.5053,B 17.4898,C -0.2766,E1 17.6324,E2 478.3248} C_DIS
LIN {X 113.9085,Y -65.6872,Z 159,A -31.3741,B 17.4898,C -0.2727,E1 17.6298,E2 480.1924} C_DIS
LIN {X 111.6985,Y -69.3785,Z 159,A -33.0513,B 17.4898,C -0.2752,E1 17.6274,E2 481.8485} C_DIS
LIN {X 109.671,Y -72.5414,Z 159,A -34.8399,B 17.49,C -0.265,E1 17.6247,E2 483.6577} C_DIS
LIN {X 106.4161,Y -77.2368,Z 159,A -37.3505,B 17.49,C -0.2577,E1 17.6206,E2 486.1743} C_DIS
LIN {X 102.8623,Y -81.91,Z 159,A -39.8282,B 17.4901,C -0.2543,E1 17.6164,E2 488.646} C_DIS
LIN {X 97.5356,Y -88.186,Z 159,A -43.1639,B 17.4901,C -0.2551,E1 17.6104,E2 491.9565} C_DIS
LIN {X 93.2788,Y -92.6767,Z 159,A -45.7331,B 17.4901,C -0.2536,E1 17.6055,E2 494.514} C_DIS
LIN {X 88.5024,Y -97.2485,Z 159,A -48.7938,B 17.4903,C -0.2402,E1 17.5992,E2 497.6004} C_DIS
LIN {X 84.8794,Y -100.4268,Z 159,A -50.9198,B 17.4903,C -0.2347,E1 17.5947,E2 499.7323} C_DIS
LIN {X 80.0311,Y -104.331,Z 159,A -53.799,B 17.4905,C -0.2228,E1 17.5884,E2 502.6349} C_DIS
LIN {X 77.3981,Y -106.2992,Z 159,A -55.1862,B 17.4905,C -0.2217,E1 17.5853,E2 504.0185} C_DIS
LIN {X 73.8892,Y -108.7674,Z 159,A -57.0152,B 17.4905,C -0.2197,E1 17.581,E2 505.8449} C_DIS
LIN {X 68.0774,Y -112.4961,Z 159,A -59.9803,B 17.4906,C -0.216,E1 17.5741,E2 508.8082} C_DIS
LIN {X 64.3611,Y -114.6628,Z 159,A -61.8684,B 17.4906,C -0.2123,E1 17.5695,E2 510.7001} C_DIS
LIN {X 60.3093,Y -116.8448,Z 159,A -64.1595,B 17.4908,C -0.1985,E1 17.5637,E2 513.0275} C_DIS
LIN {X 57.1039,Y -118.443,Z 159,A -65.1832,B 17.4906,C -0.2162,E1 17.5613,E2 513.9885} C_DIS
LIN {X 53.747,Y -120.0027,Z 159,A -66.9734,B 17.4907,C -0.2072,E1 17.5567,E2 515.8016} C_DIS
LIN {X 50.3798,Y -121.4552,Z 159,A -68.5311,B 17.4907,C -0.2065,E1 17.5527,E2 517.3561} C_DIS
LIN {X 46.5074,Y -122.9904,Z 159,A -70.42,B 17.4907,C -0.2015,E1 17.5478,E2 519.2556} C_DIS
LIN {X 43.1433,Y -124.2098,Z 159,A -71.9479,B 17.4907,C -0.2008,E1 17.5437,E2 520.7812} C_DIS
LIN {X 39.1617,Y -125.5241,Z 159,A -73.8702,B 17.4908,C -0.1952,E1 17.5386,E2 522.7166} C_DIS
LIN {X 33.5936,Y -127.1259,Z 159,A -76.229,B 17.4908,C -0.1989,E1 17.5323,E2 525.0576} C_DIS
LIN {X 29.8622,Y -128.0549,Z 159,A -78.3164,B 17.491,C -0.1823,E1 17.5265,E2 527.1956} C_DIS
LIN {X 26.2004,Y -128.8526,Z 159,A -79.6681,B 17.4909,C -0.1913,E1 17.5229,E2 528.515} C_DIS
LIN {X 22.6325,Y -129.5281,Z 159,A -81.1887,B 17.4909,C -0.1924,E1 17.5187,E2 530.0294} C_DIS
LIN {X 18.706,Y -130.1522,Z 159,A -82.8366,B 17.4909,C -0.1944,E1 17.5142,E2 531.6683} C_DIS
LIN {X 15.2808,Y -130.5989,Z 159,A -84.3131,B 17.4909,C -0.1946,E1 17.5101,E2 533.1424} C_DIS
LIN {X 11.4583,Y -130.99,Z 159,A -86.0681,B 17.4909,C -0.1909,E1 17.5052,E2 534.9081} C_DIS
LIN {X 7.7681,Y -131.2603,Z 159,A -87.723,B 17.4909,C -0.1887,E1 17.5006,E2 536.5691} C_DIS
LIN {X 3.4482,Y -131.4446,Z 159,A -89.5304,B 17.4909,C -0.1909,E1 17.4955,E2 538.3683} C_DIS
LIN {X 0.9129,Y -131.485,Z 159,A -90.5204,B 17.4909,C -0.1949,E1 17.4928,E2 539.345} C_DIS
Enddeposition()
LIN {X 0.9129,Y -131.485,Z 159,A -90.5204,B 17.4909,C -0.1949,E1 17.4928,E2 539.345} C_DIS
Startdeposition()
$VEL.CP = VEL_PRINT
LIN {X 2.4689,Y -130.5387,Z 159,A -88.3234,B 14.7758,C 0.0231,E1 14.7809,E2 537.7887} C_DIS
LIN {X 6.539,Y -130.3978,Z 159,A -86.6339,B 14.7758,C 0.0256,E1 14.7856,E2 536.11} C_DIS
LIN {X 10.6995,Y -130.1228,Z 159,A -84.764,B 14.7758,C 0.0237,E1 14.7908,E2 534.2342} C_DIS
LIN {X 14.8726,Y -129.7131,Z 159,A -82.9309,B 14.7758,C 0.0231,E1 14.7959,E2 532.4008} C_DIS
LIN {X 18.3964,Y -129.259,Z 159,A -81.4327,B 14.7758,C 0.0241,E1 14.8001,E2 530.9089} C_DIS
LIN {X 21.7164,Y -128.743,Z 159,A -79.8926,B 14.7758,C 0.0211,E1 14.8043,E2 529.3599} C_DIS
LIN {X 30.2826,Y -127.0014,Z 159,A -76.1219,B 14.7758,C 0.0202,E1 14.8146,E2 525.5945} C_DIS
LIN {X 36.8099,Y -125.265,Z 159,A -73.2022,B 14.7758,C 0.0189,E1 14.8225,E2 522.6779} C_DIS
LIN {X 42.521,Y -123.4434,Z 159,A -70.6693,B 14.7758,C 0.0191,E1 14.8292,E2 520.1546} C_DIS
LIN {X 45.4458,Y -122.3971,Z 159,A -69.1049,B 14.7758,C 0.0111,E1 14.8334,E2 518.5648} C_DIS
LIN {X 49.1763,Y -120.9466,Z 159,A -67.4403,B 14.7758,C 0.0119,E1 14.8376,E2 516.9097} C_DIS
LIN {X 52.8865,Y -119.3711,Z 159,A -65.6447,B 14.7758,C 0.0087,E1 14.8423,E2 515.1093} C_DIS
LIN {X 56.5684,Y -117.6704,Z 159,A -63.1571,B 14.7758,C -0.0167,E1 14.8488,E2 512.5341} C_DIS
LIN {X 61.6493,Y -115.0918,Z 159,A -61.354,B 14.7758,C 0.002,E1 14.853,E2 510.8133} C_DIS
LIN {X 65.3737,Y -113.0178,Z 159,A -59.5473,B 14.7758,C 0.0011,E1 14.8574,E2 509.0123} C_DIS
LIN {X 68.4752,Y -111.1663,Z 159,A -57.818,B 14.7758,C -0.0063,E1 14.8615,E2 507.2639} C_DIS
LIN {X 72.3821,Y -108.6627,Z 159,A -55.8884,B 14.7758,C -0.0064,E1 14.866,E2 505.345} C_DIS
LIN {X 75.7094,Y -106.3715,Z 159,A -54.0881,B 14.7758,C -0.0106,E1 14.8701,E2 503.5395} C_DIS
LIN {X 79.4434,Y -103.6123,Z 159,A -52.2569,B 14.7758,C -0.0078,E1 14.8742,E2 501.7308} C_DIS
LIN {X 82.6305,Y -101.0888,Z 159,A -50.3479,B 14.7758,C -0.0155,E1 14.8784,E2 499.8048} C_DIS
LIN {X 86.025,Y -98.2165,Z 159,A -48.4238,B 14.7758,C -0.0186,E1 14.8825,E2 497.8816} C_DIS
LIN {X 89.5438,Y -95.0192,Z 159,A -46.0147,B 14.7758,C -0.0338,E1 14.8875,E2 495.4311} C_DIS
LIN {X 92.2325,Y -92.412,Z 159,A -44.6908,B 14.7758,C -0.0269,E1 14.89,E2 494.1439} C_DIS
LIN {X 95.2878,Y -89.2587,Z 159,A -42.89,B 14.7758,C -0.0271,E1 14.8935,E2 492.3558} C_DIS
LIN {X 98.3401,Y -85.8833,Z 159,A -40.5737,B 14.7758,C -0.0424,E1 14.8978,E2 489.9986} C_DIS
LIN {X 100.4825,Y -83.3668,Z 159,A -39.3446,B 14.7758,C -0.0385,E1 14.9,E2 488.7944} C_DIS
LIN {X 103.2626,Y -79.8972,Z 159,A -37.4747,B 14.7758,C -0.0406,E1 14.9032,E2 486.9318} C_DIS
LIN {X 106.3579,Y -75.7283,Z 159,A -35.1937,B 14.7758,C -0.0464,E1 14.907,E2 484.6476} C_DIS
LIN {X 108.7197,Y -72.2966,Z 159,A -33.3725,B 14.7758,C -0.0509,E1 14.9098,E2 482.8249} C_DIS
LIN {X 110.9208,Y -68.8718,Z 159,A -31.6162,B 14.7758,C -0.0546,E1 14.9124,E2 481.07} C_DIS
LIN {X 113.1804,Y -65.0928,Z 159,A -29.6544,B 14.7757,C -0.0607,E1 14.9152,E2 479.1021} C_DIS
LIN {X 115.1775,Y -61.4898,Z 159,A -27.8722,B 14.7757,C -0.0648,E1 14.9176,E2 477.3206} C_DIS
LIN {X 116.9466,Y -58.0501,Z 159,A -26.4886,B 14.7757,C -0.059,E1 14.9193,E2 475.9723} C_DIS
LIN {X 118.9713,Y -53.7803,Z 159,A -23.5267,B 14.7755,C -0.0946,E1 14.9229,E2 472.9006} C_DIS
LIN {X 121.0486,Y -48.9233,Z 159,A -21.2353,B 14.7755,C -0.1003,E1 14.9253,E2 470.6094} C_DIS
LIN {X 122.9455,Y -43.9405,Z 159,A -19.6054,B 14.7755,C -0.0831,E1 14.9268,E2 469.0623} C_DIS
LIN {X 124.2939,Y -39.9668,Z 159,A -17.7689,B 14.7755,C -0.0883,E1 14.9284,E2 467.224} C_DIS
LIN {X 125.2573,Y -36.836,Z 159,A -16.0407,B 14.7755,C -0.1023,E1 14.9298,E2 465.4589} C_DIS
LIN {X 126.1756,Y -33.5558,Z 159,A -14.8356,B 14.7755,C -0.0969,E1 14.9306,E2 464.2867} C_DIS
LIN {X 127.2461,Y -29.2358,Z 159,A -13.2247,B 14.7755,C -0.0913,E1 14.9317,E2 462.7143} C_DIS
LIN {X 128.0389,Y -25.5455,Z 159,A -11.4563,B 14.7755,C -0.0999,E1 14.9327,E2 460.9304} C_DIS
LIN {X 129.2001,Y -18.8089,Z 159,A -8.2946,B 14.7754,C -0.1143,E1 14.9342,E2 457.7457} C_DIS
LIN {X 129.5853,Y -15.9442,Z 159,A -6.8921,B 14.7754,C -0.1226,E1 14.9346,E2 456.3255} C_DIS
LIN {X 130.0844,Y -11.1546,Z 159,A -4.9964,B 14.7754,C -0.1216,E1 14.9351,E2 454.4531} C_DIS
LIN {X 130.3514,Y -7.431,Z 159,A -3.2825,B 14.7753,C -0.1291,E1 14.9354,E2 452.7282} C_DIS
LIN {X 130.5139,Y -3.5345,Z 159,A -1.6502,B 14.7753,C -0.1316,E1 14.9356,E2 451.1032} C_DIS
LIN {X 130.5605,Y 0.7161,Z 159,A 0.1727,B 14.7753,C -0.1358,E1 14.9356,E2 449.2832} C_DIS
LIN {X 130.4791,Y 4.6639,Z 159,A 1.9391,B 14.7751,C -0.1422,E1 14.9355,E2 447.5106} C_DIS
LIN {X 130.276,Y 8.655,Z 159,A 3.7204,B 14.7751,C -0.1483,E1 14.9352,E2 445.724} C_DIS
LIN {X 130.0009,Y 12.093,Z 159,A 5.1306,B 14.7751,C -0.1494,E1 14.9348,E2 444.3242} C_DIS
LIN {X 129.6249,Y 15.6121,Z 159,A 6.6508,B 14.7751,C -0.153,E1 14.9343,E2 442.8062} C_DIS
LIN {X 129.1218,Y 19.3465,Z 159,A 8.429,B 14.7749,C -0.162,E1 14.9336,E2 441.0112} C_DIS
LIN {X 128.6247,Y 22.4129,Z 159,A 9.992,B 14.7749,C -0.1727,E1 14.9329,E2 439.4229} C_DIS
LIN {X 127.98,Y 25.8353,Z 159,A 11.3985,B 14.7749,C -0.1731,E1 14.9321,E2 438.0293} C_DIS
LIN {X 126.6754,Y 31.6211,Z 159,A 13.814,B 14.7749,C -0.1744,E1 14.9306,E2 435.6333} C_DIS
LIN {X 125.7874,Y 34.9833,Z 159,A 15.2349,B 14.7748,C -0.1753,E1 14.9295,E2 434.2233} C_DIS
LIN {X 124.8427,Y 38.2173,Z 159,A 16.872,B 14.7747,C -0.1848,E1 14.9282,E2 432.5658} C_DIS
LIN {X 123.4524,Y 42.4951,Z 159,A 18.6368,B 14.7747,C -0.1834,E1 14.9266,E2 430.824} C_DIS
LIN {X 122.3435,Y 45.5889,Z 159,A 20.0575,B 14.7747,C -0.1868,E1 14.9253,E2 429.4043} C_DIS
LIN {X 121.3454,Y 48.1868,Z 159,A 21.2782,B 14.7747,C -0.1901,E1 14.924,E2 428.1826} C_DIS
LIN {X 119.8632,Y 51.7593,Z 159,A 22.9441,B 14.7746,C -0.1937,E1 14.9222,E2 426.5188} C_DIS
LIN {X 118.4871,Y 54.8363,Z 159,A 24.3913,B 14.7746,C -0.1966,E1 14.9206,E2 425.074} C_DIS
LIN {X 117.119,Y 57.7005,Z 159,A 25.7617,B 14.7745,C -0.1996,E1 14.9189,E2 423.705} C_DIS
LIN {X 115.6946,Y 60.5064,Z 159,A 27.1249,B 14.7745,C -0.2027,E1 14.9171,E2 422.3428} C_DIS
LIN {X 113.8629,Y 63.8903,Z 159,A 28.9019,B 14.7744,C -0.2099,E1 14.9147,E2 420.554} C_DIS
LIN {X 111.8155,Y 67.4096,Z 159,A 30.7201,B 14.7743,C -0.2155,E1 14.9121,E2 418.7306} C_DIS
LIN {X 109.457,Y 71.1751,Z 159,A 32.5632,B 14.7743,C -0.2168,E1 14.9094,E2 416.8986} C_DIS
LIN {X 107.3821,Y 74.2694,Z 159,A 34.2106,B 14.7742,C -0.2212,E1 14.9068,E2 415.2485} C_DIS
LIN {X 105.0209,Y 77.5722,Z 159,A 35.9986,B 14.7742,C -0.2256,E1 14.9039,E2 413.4586} C_DIS
LIN {X 102.4457,Y 80.9428,Z 159,A 37.9149,B 14.774,C -0.2317,E1 14.9006,E2 411.5346} C_DIS
LIN {X 99.7904,Y 84.1946,Z 159,A 39.7488,B 14.774,C -0.2356,E1 14.8973,E2 409.7005} C_DIS
LIN {X 97.4522,Y 86.8901,Z 159,A 41.9245,B 14.7736,C -0.2589,E1 14.8931,E2 407.4513} C_DIS
LIN {X 93.6748,Y 90.9494,Z 159,A 43.6795,B 14.7739,C -0.2419,E1 14.8899,E2 405.7757} C_DIS
LIN {X 90.5109,Y 94.0993,Z 159,A 45.6661,B 14.7738,C -0.2468,E1 14.8859,E2 403.7849} C_DIS
LIN {X 87.2405,Y 97.1383,Z 159,A 47.5829,B 14.7738,C -0.2493,E1 14.8819,E2 401.8721} C_DIS
LIN {X 84.3042,Y 99.6978,Z 159,A 49.1485,B 14.7738,C -0.2479,E1 14.8787,E2 400.3227} C_DIS
LIN {X 78.05,Y 104.6658,Z 159,A 52.7318,B 14.7736,C -0.2566,E1 14.8708,E2 396.729} C_DIS
LIN {X 74.5158,Y 107.2106,Z 159,A 54.5766,B 14.7736,C -0.2576,E1 14.8666,E2 394.8914} C_DIS
LIN {X 71.2368,Y 109.417,Z 159,A 56.3845,B 14.7736,C -0.2627,E1 14.8623,E2 393.0745} C_DIS
LIN {X 67.3402,Y 111.8575,Z 159,A 58.373,B 14.7735,C -0.2648,E1 14.8576,E2 391.0889} C_DIS
LIN {X 63.5948,Y 114.0289,Z 159,A 60.2992,B 14.7735,C -0.2683,E1 14.8529,E2 389.1593} C_DIS
LIN {X 59.7831,Y 116.0714,Z 159,A 62.0845,B 14.7735,C -0.2673,E1 14.8485,E2 387.3869} C_DIS
LIN {X 56.6059,Y 117.6525,Z 159,A 63.6423,B 14.7735,C -0.2692,E1 14.8446,E2 385.8288} C_DIS
LIN {X 53.6573,Y 119.0263,Z 159,A 65.0693,B 14.7734,C -0.2709,E1 14.841,E2 384.4017} C_DIS
LIN {X 50.5643,Y 120.3726,Z 159,A 66.5268,B 14.7734,C -0.2718,E1 14.8373,E2 382.9469} C_DIS
LIN {X 47.5654,Y 121.5888,Z 159,A 67.9648,B 14.7734,C -0.2738,E1 14.8335,E2 381.5068} C_DIS
LIN {X 44.3941,Y 122.782,Z 159,A 69.414,B 14.7734,C -0.274,E1 14.8297,E2 380.062} C_DIS
LIN {X 41.384,Y 123.8291,Z 159,A 70.8483,B 14.7733,C -0.2764,E1 14.8259,E2 378.6237} C_DIS
LIN {X 38.1375,Y 124.8671,Z 159,A 72.3525,B 14.7733,C -0.2778,E1 14.8219,E2 377.1185} C_DIS
LIN {X 34.0805,Y 126.0357,Z 159,A 74.0546,B 14.7733,C -0.2746,E1 14.8174,E2 375.4343} C_DIS
LIN {X 30.8004,Y 126.8766,Z 159,A 75.6226,B 14.7733,C -0.278,E1 14.8131,E2 373.8569} C_DIS
LIN {X 27.7357,Y 127.5816,Z 159,A 77.0337,B 14.7733,C -0.2797,E1 14.8093,E2 372.4425} C_DIS
LIN {X 24.5942,Y 128.2241,Z 159,A 78.7006,B 14.7731,C -0.2883,E1 14.8046,E2 370.7456} C_DIS
LIN {X 19.7863,Y 129.0537,Z 159,A 80.4756,B 14.7733,C -0.2781,E1 14.7999,E2 369.014} C_DIS
LIN {X 14.28,Y 129.7787,Z 159,A 83.0112,B 14.7732,C -0.2817,E1 14.7928,E2 366.4677} C_DIS
LIN {X 10.7993,Y 130.1144,Z 159,A 84.5706,B 14.7732,C -0.2827,E1 14.7885,E2 364.906} C_DIS
LIN {X 6.7716,Y 130.3861,Z 159,A 86.3092,B 14.7732,C -0.2819,E1 14.7836,E2 363.1719} C_DIS
LIN {X 2.8832,Y 130.5318,Z 159,A 88.1023,B 14.7732,C -0.2844,E1 14.7786,E2 361.3698} C_DIS
LIN {X -1.4401,Y 130.5558,Z 159,A 89.9611,B 14.7732,C -0.2831,E1 14.7734,E2 359.5163} C_DIS
LIN {X -5.2465,Y 130.4563,Z 159,A 91.642,B 14.7732,C -0.2831,E1 14.7687,E2 357.8351} C_DIS
LIN {X -9.3949,Y 130.2232,Z 159,A 93.4011,B 14.7732,C -0.2807,E1 14.7638,E2 356.0844} C_DIS
LIN {X -12.7844,Y 129.9346,Z 159,A 94.9863,B 14.7732,C -0.2828,E1 14.7594,E2 354.4893} C_DIS
LIN {X -15.7945,Y 129.6031,Z 159,A 96.5203,B 14.7731,C -0.2882,E1 14.7551,E2 352.9323} C_DIS
LIN {X -19.0273,Y 129.1689,Z 159,A 97.6101,B 14.7733,C -0.2775,E1 14.7522,E2 351.8833} C_DIS
LIN {X -22.8409,Y 128.5481,Z 159,A 99.8561,B 14.773,C -0.2926,E1 14.7458,E2 349.5741} C_DIS
LIN {X -27.0446,Y 127.7308,Z 159,A 101.2907,B 14.7733,C -0.2783,E1 14.7421,E2 348.1929} C_DIS
LIN {X -33.2766,Y 126.2501,Z 159,A 104.0519,B 14.7733,C -0.2745,E1 14.7346,E2 345.4396} C_DIS
LIN {X -36.5194,Y 125.35,Z 159,A 105.5442,B 14.7733,C -0.2736,E1 14.7306,E2 343.9467} C_DIS
LIN {X -39.7029,Y 124.3782,Z 159,A 106.8665,B 14.7734,C -0.2682,E1 14.7271,E2 342.6415} C_DIS
LIN {X -43.9777,Y 122.9321,Z 159,A 108.9587,B 14.7734,C -0.2693,E1 14.7216,E2 340.5382} C_DIS
LIN {X -46.7216,Y 121.9169,Z 159,A 110.2682,B 14.7734,C -0.2686,E1 14.7181,E2 339.2269} C_DIS
LIN {X -50.6873,Y 120.3212,Z 159,A 112.4369,B 14.7734,C -0.2746,E1 14.7124,E2 337.0257} C_DIS
LIN {X -54.9672,Y 118.4266,Z 159,A 114.298,B 14.7734,C -0.2664,E1 14.7078,E2 335.189} C_DIS
LIN {X -58.7432,Y 116.6008,Z 159,A 116.0121,B 14.7736,C -0.2602,E1 14.7035,E2 333.4914} C_DIS
LIN {X -61.7051,Y 115.0619,Z 159,A 117.9999,B 14.7734,C -0.2728,E1 14.6985,E2 331.4443} C_DIS
LIN {X -65.1689,Y 113.1363,Z 159,A 119.4049,B 14.7736,C -0.2606,E1 14.6952,E2 330.0799} C_DIS
LIN {X -68.9626,Y 110.8643,Z 159,A 121.3237,B 14.7736,C -0.2568,E1 14.6906,E2 328.1657} C_DIS
LIN {X -72.6156,Y 108.5068,Z 159,A 123.1739,B 14.7737,C -0.2519,E1 14.6863,E2 326.3242} C_DIS
LIN {X -75.3177,Y 106.6489,Z 159,A 124.7054,B 14.7737,C -0.2519,E1 14.6828,E2 324.7835} C_DIS
LIN {X -78.9624,Y 103.9799,Z 159,A 126.7344,B 14.7737,C -0.2494,E1 14.6782,E2 322.7514} C_DIS
LIN {X -82.3292,Y 101.3349,Z 159,A 128.6451,B 14.7738,C -0.2466,E1 14.6741,E2 320.8391} C_DIS
LIN {X -85.77,Y 98.439,Z 159,A 130.5899,B 14.7738,C -0.2418,E1 14.6699,E2 318.8999} C_DIS
LIN {X -89.1271,Y 95.4103,Z 159,A 132.3423,B 14.774,C -0.2313,E1 14.6664,E2 317.1767} C_DIS
LIN {X -91.8202,Y 92.8216,Z 159,A 134.268,B 14.774,C -0.2356,E1 14.6625,E2 315.2198} C_DIS
LIN {X -94.9049,Y 89.665,Z 159,A 136.2091,B 14.774,C -0.2314,E1 14.6587,E2 313.2806} C_DIS
LIN {X -97.831,Y 86.4629,Z 159,A 138.1159,B 14.7741,C -0.2271,E1 14.6552,E2 311.3757} C_DIS
LIN {X -100.773,Y 83.0159,Z 159,A 140.1297,B 14.7741,C -0.223,E1 14.6516,E2 309.3614} C_DIS
LIN {X -103.4926,Y 79.5998,Z 159,A 142.0911,B 14.7742,C -0.2196,E1 14.6482,E2 307.3972} C_DIS
LIN {X -106.2079,Y 75.9383,Z 159,A 144.061,B 14.7743,C -0.2138,E1 14.645,E2 305.4334} C_DIS
LIN {X -108.7548,Y 72.2441,Z 159,A 146.0524,B 14.7743,C -0.2094,E1 14.6418,E2 303.4419} C_DIS
LIN {X -110.9745,Y 68.7854,Z 159,A 147.8754,B 14.7744,C -0.2052,E1 14.6391,E2 301.6189} C_DIS
LIN {X -113.2217,Y 65.0209,Z 159,A 149.6361,B 14.7745,C -0.1957,E1 14.6367,E2 299.8798} C_DIS
LIN {X -115.2704,Y 61.3142,Z 159,A 151.6905,B 14.7745,C -0.196,E1 14.6339,E2 297.8049} C_DIS
LIN {X -116.71,Y 58.5287,Z 159,A 153.1802,B 14.7745,C -0.1953,E1 14.632,E2 296.3039} C_DIS
LIN {X -118.2824,Y 55.2791,Z 159,A 154.5194,B 14.7747,C -0.1843,E1 14.6304,E2 294.9952} C_DIS
LIN {X -119.4721,Y 52.6606,Z 159,A 155.952,B 14.7747,C -0.1853,E1 14.6288,E2 293.5445} C_DIS
LIN {X -120.8928,Y 49.3097,Z 159,A 157.5563,B 14.7747,C -0.181,E1 14.6271,E2 291.9414} C_DIS
LIN {X -122.0286,Y 46.4298,Z 159,A 158.9591,B 14.7747,C -0.1784,E1 14.6257,E2 290.5352} C_DIS
LIN {X -123.2879,Y 42.9697,Z 159,A 160.364,B 14.7749,C -0.1681,E1 14.6244,E2 289.157} C_DIS
LIN {X -124.2277,Y 40.174,Z 159,A 161.7421,B 14.7749,C -0.1666,E1 14.6232,E2 287.7708} C_DIS
LIN {X -125.2211,Y 36.9596,Z 159,A 163.2421,B 14.7749,C -0.1629,E1 14.622,E2 286.27} C_DIS
LIN {X -126.105,Y 33.8207,Z 159,A 164.6246,B 14.7749,C -0.1574,E1 14.6209,E2 284.8951} C_DIS
LIN {X -126.8659,Y 30.8445,Z 159,A 166.1568,B 14.7749,C -0.1584,E1 14.6199,E2 283.3432} C_DIS
LIN {X -127.823,Y 26.6068,Z 159,A 168.1132,B 14.775,C -0.154,E1 14.6187,E2 281.3835} C_DIS
LIN {X -128.4398,Y 23.4462,Z 159,A 169.6261,B 14.775,C -0.1525,E1 14.618,E2 279.8607} C_DIS
LIN {X -129.1787,Y 18.9587,Z 159,A 171.5173,B 14.7751,C -0.1437,E1 14.6171,E2 277.9842} C_DIS
LIN {X -129.6653,Y 15.2731,Z 159,A 173.1085,B 14.7751,C -0.1378,E1 14.6166,E2 276.3998} C_DIS
LIN {X -130.0553,Y 11.4992,Z 159,A 174.7846,B 14.7752,C -0.133,E1 14.6161,E2 274.7246} C_DIS
LIN {X -130.4092,Y 6.3139,Z 159,A 177.0333,B 14.7752,C -0.1253,E1 14.6158,E2 272.4825} C_DIS
LIN {X -130.5637,Y 0.0469,Z 159,A -179.87,B 14.7752,C -0.1263,E1 14.6156,E2 269.3488} C_DIS
LIN {X -130.4077,Y -6.3431,Z 159,A -177.4327,B 14.7754,C -0.108,E1 14.6158,E2 266.958} C_DIS
LIN {X -129.8873,Y -13.2705,Z 159,A -174.1218,B 14.7754,C -0.1058,E1 14.6166,E2 263.6202} C_DIS
LIN {X -129.1843,Y -18.9192,Z 159,A -171.6936,B 14.7755,C -0.0966,E1 14.6175,E2 261.203} C_DIS
LIN {X -128.6735,Y -22.1331,Z 159,A -170.2012,B 14.7755,C -0.0941,E1 14.6182,E2 259.7047} C_DIS
LIN {X -127.9495,Y -25.985,Z 159,A -168.1839,B 14.7755,C -0.0971,E1 14.6193,E2 257.6543} C_DIS
LIN {X -127.2593,Y -29.1783,Z 159,A -167.0889,B 14.7755,C -0.0838,E1 14.6199,E2 256.6007} C_DIS
LIN {X -126.6076,Y -31.8882,Z 159,A -165.7597,B 14.7755,C -0.0831,E1 14.6208,E2 255.2603} C_DIS
LIN {X -125.6537,Y -35.4615,Z 159,A -164.0463,B 14.7755,C -0.0809,E1 14.6221,E2 253.5381} C_DIS
LIN {X -124.4954,Y -39.3359,Z 159,A -162.3915,B 14.7756,C -0.0726,E1 14.6234,E2 251.8992} C_DIS
LIN {X -123.4022,Y -42.6399,Z 159,A -160.8956,B 14.7756,C -0.0675,E1 14.6248,E2 250.4084} C_DIS
LIN {X -121.4129,Y -48.0181,Z 159,A -158.1554,B 14.7756,C -0.0665,E1 14.6275,E2 247.6445} C_DIS
LIN {X -119.9339,Y -51.596,Z 159,A -156.6612,B 14.7757,C -0.0564,E1 14.6291,E2 246.1759} C_DIS
LIN {X -118.5564,Y -54.6865,Z 159,A -154.5751,B 14.7757,C -0.0688,E1 14.6316,E2 244.0202} C_DIS
LIN {X -116.6681,Y -58.611,Z 159,A -153.0945,B 14.7757,C -0.0519,E1 14.6334,E2 242.5923} C_DIS
LIN {X -115.0609,Y -61.7068,Z 159,A -151.5312,B 14.7757,C -0.0489,E1 14.6354,E2 241.0264} C_DIS
LIN {X -113.1608,Y -65.1265,Z 159,A -149.7053,B 14.7757,C -0.0475,E1 14.638,E2 239.1892} C_DIS
LIN {X -110.7699,Y -69.1142,Z 159,A -147.7426,B 14.7757,C -0.0402,E1 14.6408,E2 237.2373} C_DIS
LIN {X -106.9694,Y -74.8626,Z 159,A -144.633,B 14.7757,C -0.0353,E1 14.6457,E2 234.1199} C_DIS
LIN {X -104.5017,Y -78.2704,Z 159,A -142.8145,B 14.7757,C -0.0302,E1 14.6487,E2 232.306} C_DIS
LIN {X -102.6366,Y -80.6998,Z 159,A -141.389,B 14.7757,C -0.0294,E1 14.6512,E2 230.8717} C_DIS
LIN {X -99.7523,Y -84.2399,Z 159,A -139.3979,B 14.7757,C -0.0246,E1 14.6547,E2 228.8834} C_DIS
LIN {X -97.3009,Y -87.059,Z 159,A -137.5609,B 14.7757,C -0.0266,E1 14.6582,E2 227.0239} C_DIS
LIN {X -95.0698,Y -89.4901,Z 159,A -136.3194,B 14.7758,C -0.0177,E1 14.6605,E2 225.8078} C_DIS
LIN {X -91.9999,Y -92.6431,Z 159,A -134.558,B 14.7758,C -0.009,E1 14.6639,E2 224.0675} C_DIS
LIN {X -88.534,Y -95.961,Z 159,A -132.2448,B 14.7758,C -0.0107,E1 14.6686,E2 221.7307} C_DIS
LIN {X -85.2062,Y -98.9274,Z 159,A -130.5065,B 14.7758,C -0.0009,E1 14.6722,E2 220.0192} C_DIS
LIN {X -80.2174,Y -103.0145,Z 159,A -127.4423,B 14.7758,C -0.0024,E1 14.6789,E2 216.9285} C_DIS
LIN {X -76.9181,Y -105.501,Z 159,A -125.643,B 14.7758,C 0.001,E1 14.683,E2 215.1314} C_DIS
LIN {X -73.6348,Y -107.8181,Z 159,A -123.8205,B 14.7758,C 0.0021,E1 14.6872,E2 213.3024} C_DIS
LIN {X -70.8336,Y -109.6788,Z 159,A -122.5387,B 14.7758,C 0.0099,E1 14.6901,E2 212.0442} C_DIS
LIN {X -65.9422,Y -112.6872,Z 159,A -119.8131,B 14.7758,C 0.0076,E1 14.6967,E2 209.2947} C_DIS
LIN {X -62.1223,Y -114.8377,Z 159,A -117.865,B 14.7758,C 0.0095,E1 14.7015,E2 207.344} C_DIS
LIN {X -58.4801,Y -116.7345,Z 159,A -116.0169,B 14.7758,C 0.0103,E1 14.7061,E2 205.4906} C_DIS
LIN {X -54.8676,Y -118.4727,Z 159,A -114.4336,B 14.7758,C 0.0175,E1 14.71,E2 203.9283} C_DIS
LIN {X -51.7593,Y -119.8633,Z 159,A -112.987,B 14.7758,C 0.0205,E1 14.7137,E2 202.4876} C_DIS
LIN {X -49.236,Y -120.9225,Z 159,A -111.7237,B 14.7758,C 0.0199,E1 14.717,E2 201.2168} C_DIS
LIN {X -46.2595,Y -122.0924,Z 159,A -110.2446,B 14.7758,C 0.019,E1 14.7209,E2 199.7287} C_DIS
LIN {X -42.7415,Y -123.367,Z 159,A -108.6589,B 14.7758,C 0.022,E1 14.725,E2 198.1497} C_DIS
LIN {X -39.5335,Y -124.4323,Z 159,A -107.028,B 14.7758,C 0.0188,E1 14.7294,E2 196.501} C_DIS
LIN {X -35.2097,Y -125.7241,Z 159,A -105.2727,B 14.7758,C 0.0269,E1 14.734,E2 194.7724} C_DIS
LIN {X -32.157,Y -126.5393,Z 159,A -103.7889,B 14.7758,C 0.0249,E1 14.7381,E2 193.2767} C_DIS
LIN {X -29.3023,Y -127.231,Z 159,A -102.0809,B 14.7758,C 0.013,E1 14.7429,E2 191.5182} C_DIS
LIN {X -25.5093,Y -128.0463,Z 159,A -100.6723,B 14.7758,C 0.0226,E1 14.7466,E2 190.1445} C_DIS
LIN {X -21.7614,Y -128.7355,Z 159,A -99.0221,B 14.7758,C 0.0239,E1 14.7511,E2 188.4965} C_DIS
LIN {X -17.5972,Y -129.3718,Z 159,A -97.1655,B 14.7758,C 0.0242,E1 14.7563,E2 186.6385} C_DIS
LIN {X -14.072,Y -129.8011,Z 159,A -95.6656,B 14.7758,C 0.0262,E1 14.7604,E2 185.145} C_DIS
LIN {X -9.8184,Y -130.1923,Z 159,A -93.7698,B 14.7758,C 0.0258,E1 14.7657,E2 183.246} C_DIS
LIN {X -5.7623,Y -130.4362,Z 159,A -91.9592,B 14.7758,C 0.0249,E1 14.7708,E2 181.4315} C_DIS
LIN {X -1.6281,Y -130.5527,Z 159,A -90.1306,B 14.7758,C 0.0244,E1 14.7759,E2 179.6003} C_DIS
LIN {X 0.9024,Y -130.5564,Z 159,A -89.2341,B 14.7758,C 0.0307,E1 14.7783,E2 178.7288} C_DIS
Enddeposition()
LIN {X 0.9024,Y -130.5564,Z 159,A -89.2341,B 14.7758,C 0.0307,E1 14.7783,E2 178.7288} C_DIS
Startdeposition()
$VEL.CP = VEL_PRINT
LIN {X -0.0059,Y -129.6357,Z 159,A -90.2262,B 14.7758,C 0.0395,E1 14.7754,E2 179.7552} C_DIS
LIN {X -3.7359,Y -129.58,Z 159,A -91.9011,B 14.7758,C 0.0404,E1 14.7707,E2 181.4338} C_DIS
LIN {X -7.9456,Y -129.39,Z 159,A -93.7857,B 14.7758,C 0.041,E1 14.7655,E2 183.3218} C_DIS
LIN {X -12.1605,Y -129.0622,Z 159,A -95.5867,B 14.7758,C 0.0388,E1 14.7605,E2 185.1156} C_DIS
LIN {X -15.8702,Y -128.6595,Z 159,A -97.2208,B 14.7758,C 0.0381,E1 14.756,E2 186.7484} C_DIS
LIN {X -19.018,Y -128.2328,Z 159,A -98.6275,B 14.7758,C 0.0378,E1 14.7521,E2 188.1559} C_DIS
LIN {X -22.1584,Y -127.7276,Z 159,A -100.2087,B 14.7758,C 0.0424,E1 14.7477,E2 189.7581} C_DIS
LIN {X -26.3455,Y -126.9292,Z 159,A -101.926,B 14.7758,C 0.0367,E1 14.743,E2 191.4562} C_DIS
LIN {X -29.4382,Y -126.248,Z 159,A -103.3291,B 14.7758,C 0.0361,E1 14.7392,E2 192.8601} C_DIS
LIN {X -32.5152,Y -125.4911,Z 159,A -104.7339,B 14.7758,C 0.0354,E1 14.7354,E2 194.2656} C_DIS
LIN {X -35.1102,Y -124.7883,Z 159,A -105.9813,B 14.7758,C 0.0363,E1 14.732,E2 195.5201} C_DIS
LIN {X -38.6097,Y -123.7522,Z 159,A -107.5461,B 14.7758,C 0.0338,E1 14.7278,E2 197.0794} C_DIS
LIN {X -42.0017,Y -122.6413,Z 159,A -109.3117,B 14.7758,C 0.0379,E1 14.7231,E2 198.867} C_DIS
LIN {X -45.6878,Y -121.3156,Z 159,A -110.9194,B 14.7758,C 0.0328,E1 14.7189,E2 200.4604} C_DIS
LIN {X -49.0946,Y -119.979,Z 159,A -112.4927,B 14.7758,C 0.03,E1 14.7149,E2 202.0286} C_DIS
LIN {X -52.0184,Y -118.7403,Z 159,A -113.9268,B 14.7758,C 0.0294,E1 14.7112,E2 203.4662} C_DIS
LIN {X -55.4356,Y -117.1832,Z 159,A -115.5582,B 14.7758,C 0.0267,E1 14.707,E2 205.0941} C_DIS
LIN {X -58.2928,Y -115.7888,Z 159,A -116.9673,B 14.7758,C 0.0251,E1 14.7035,E2 206.5035} C_DIS
LIN {X -61.1142,Y -114.3259,Z 159,A -118.2888,B 14.7758,C 0.021,E1 14.7003,E2 207.8151} C_DIS
LIN {X -63.4156,Y -113.0653,Z 159,A -119.5483,B 14.7758,C 0.0222,E1 14.6972,E2 209.0861} C_DIS
LIN {X -66.0813,Y -111.5287,Z 159,A -121.0691,B 14.7758,C 0.0249,E1 14.6935,E2 210.6254} C_DIS
LIN {X -69.4022,Y -109.4928,Z 159,A -122.6959,B 14.7758,C 0.0197,E1 14.6896,E2 212.2408} C_DIS
LIN {X -72.8912,Y -107.2018,Z 159,A -124.5067,B 14.7758,C 0.0159,E1 14.6854,E2 214.047} C_DIS
LIN {X -75.4944,Y -105.3845,Z 159,A -125.9154,B 14.7758,C 0.0138,E1 14.6822,E2 215.4559} C_DIS
LIN {X -78.4956,Y -103.1689,Z 159,A -127.5801,B 14.7758,C 0.0114,E1 14.6785,E2 217.122} C_DIS
LIN {X -81.6484,Y -100.6922,Z 159,A -129.4114,B 14.7758,C 0.01,E1 14.6745,E2 218.9595} C_DIS
LIN {X -84.8924,Y -97.973,Z 159,A -131.4028,B 14.7758,C 0.0099,E1 14.6702,E2 220.9641} C_DIS
LIN {X -88.2225,Y -94.9847,Z 159,A -133.3279,B 14.7758,C 0.0046,E1 14.6663,E2 222.8821} C_DIS
LIN {X -91.2973,Y -92.0331,Z 159,A -135.221,B 14.7758,C 0.0011,E1 14.6625,E2 224.7754} C_DIS
LIN {X -94.1028,Y -89.1629,Z 159,A -137.0356,B 14.7758,C -0.0015,E1 14.659,E2 226.5937} C_DIS
LIN {X -96.0657,Y -87.044,Z 159,A -138.2936,B 14.7758,C -0.0047,E1 14.6566,E2 227.8489} C_DIS
LIN {X -98.8519,Y -83.8665,Z 159,A -140.1821,B 14.7758,C -0.0082,E1 14.6531,E2 229.7386} C_DIS
LIN {X -101.3087,Y -80.8818,Z 159,A -141.9244,B 14.7758,C -0.0111,E1 14.6501,E2 231.4838} C_DIS
LIN {X -103.7928,Y -77.6687,Z 159,A -143.7316,B 14.7758,C -0.0149,E1 14.647,E2 233.2911} C_DIS
LIN {X -105.9859,Y -74.6477,Z 159,A -145.2863,B 14.7758,C -0.0214,E1 14.6445,E2 234.8336} C_DIS
LIN {X -107.8005,Y -72.0023,Z 159,A -146.7058,B 14.7758,C -0.0248,E1 14.6423,E2 236.2522} C_DIS
LIN {X -109.5274,Y -69.3474,Z 159,A -148.2686,B 14.7758,C -0.0239,E1 14.6399,E2 237.8328} C_DIS
LIN {X -111.7148,Y -65.7654,Z 159,A -150.0936,B 14.7758,C -0.0293,E1 14.6373,E2 239.6528} C_DIS
LIN {X -113.571,Y -62.5061,Z 159,A -151.6686,B 14.7758,C -0.0358,E1 14.6352,E2 241.217} C_DIS
LIN {X -115.5402,Y -58.7811,Z 159,A -153.5514,B 14.7758,C -0.0401,E1 14.6327,E2 243.1004} C_DIS
LIN {X -116.9594,Y -55.9041,Z 159,A -154.9738,B 14.7758,C -0.0437,E1 14.631,E2 244.522} C_DIS
LIN {X -118.5155,Y -52.5266,Z 159,A -156.6377,B 14.7758,C -0.0476,E1 14.6291,E2 246.1869} C_DIS
LIN {X -119.7652,Y -49.6108,Z 159,A -158.0522,B 14.7758,C -0.0511,E1 14.6275,E2 247.6014} C_DIS
LIN {X -120.9432,Y -46.6651,Z 159,A -159.467,B 14.7758,C -0.0546,E1 14.6261,E2 249.0164} C_DIS
LIN {X -122.0558,Y -43.6724,Z 159,A -160.8918,B 14.7757,C -0.0582,E1 14.6247,E2 250.4414} C_DIS
LIN {X -123.0901,Y -40.666,Z 159,A -162.2927,B 14.7757,C -0.0622,E1 14.6235,E2 251.8403} C_DIS
LIN {X -124.0535,Y -37.625,Z 159,A -163.7335,B 14.7757,C -0.0654,E1 14.6223,E2 253.2833} C_DIS
LIN {X -124.9387,Y -34.5726,Z 159,A -165.1517,B 14.7757,C -0.0691,E1 14.6212,E2 254.7016} C_DIS
LIN {X -125.7488,Y -31.4995,Z 159,A -166.5694,B 14.7757,C -0.0728,E1 14.6202,E2 256.1193} C_DIS
LIN {X -126.4834,Y -28.4079,Z 159,A -167.9882,B 14.7757,C -0.0765,E1 14.6193,E2 257.5382} C_DIS
LIN {X -127.1461,Y -25.2794,Z 159,A -169.3727,B 14.7756,C -0.0814,E1 14.6185,E2 258.9178} C_DIS
LIN {X -127.6302,Y -22.7023,Z 159,A -170.6503,B 14.7756,C -0.0817,E1 14.6179,E2 260.2077} C_DIS
LIN {X -128.3627,Y -18.1087,Z 159,A -172.6778,B 14.7756,C -0.0885,E1 14.6171,E2 262.2296} C_DIS
LIN {X -128.8447,Y -14.2865,Z 159,A -174.5183,B 14.7756,C -0.0899,E1 14.6164,E2 264.0839} C_DIS
LIN {X -129.2443,Y -10.0596,Z 159,A -176.4291,B 14.7756,C -0.0946,E1 14.616,E2 265.9965} C_DIS
LIN {X -129.5002,Y -5.9126,Z 159,A -178.2856,B 14.7755,C -0.0996,E1 14.6157,E2 267.8531} C_DIS
LIN {X -129.6154,Y -2.1831,Z 159,A -179.8694,B 14.7755,C -0.1063,E1 14.6157,E2 269.4273} C_DIS
LIN {X -129.6265,Y 1.5126,Z 159,A 178.3747,B 14.7755,C -0.108,E1 14.6157,E2 271.1954} C_DIS
LIN {X -129.5054,Y 5.808,Z 159,A 176.464,B 14.7754,C -0.1134,E1 14.6158,E2 273.105} C_DIS
LIN {X -129.2401,Y 10.1173,Z 159,A 174.5556,B 14.7754,C -0.1191,E1 14.6162,E2 275.011} C_DIS
LIN {X -128.9025,Y 13.7495,Z 159,A 172.9755,B 14.7753,C -0.1248,E1 14.6166,E2 276.5854} C_DIS
LIN {X -128.4554,Y 17.4484,Z 159,A 171.4107,B 14.7753,C -0.1319,E1 14.6172,E2 278.1388} C_DIS
LIN {X -127.9904,Y 20.5882,Z 159,A 169.9685,B 14.7752,C -0.1351,E1 14.6178,E2 279.5838} C_DIS
LIN {X -127.3405,Y 24.2743,Z 159,A 168.2316,B 14.7752,C -0.1379,E1 14.6187,E2 281.3278} C_DIS
LIN {X -126.6063,Y 27.8558,Z 159,A 166.6792,B 14.7752,C -0.1443,E1 14.6196,E2 282.871} C_DIS
LIN {X -125.8831,Y 30.9619,Z 159,A 165.255,B 14.7751,C -0.1481,E1 14.6205,E2 284.2951} C_DIS
LIN {X -125.0871,Y 34.0363,Z 159,A 163.857,B 14.7751,C -0.1524,E1 14.6215,E2 285.6905} C_DIS
LIN {X -124.2161,Y 37.0899,Z 159,A 162.4159,B 14.7751,C -0.1555,E1 14.6226,E2 287.1341} C_DIS
LIN {X -123.2706,Y 40.1207,Z 159,A 160.9961,B 14.775,C -0.1591,E1 14.6238,E2 288.5539} C_DIS
LIN {X -122.4011,Y 42.6946,Z 159,A 159.7289,B 14.775,C -0.1608,E1 14.625,E2 289.8271} C_DIS
LIN {X -121.3107,Y 45.7009,Z 159,A 158.3018,B 14.775,C -0.1645,E1 14.6264,E2 291.2539} C_DIS
LIN {X -119.9743,Y 49.1062,Z 159,A 156.7179,B 14.7748,C -0.1699,E1 14.628,E2 292.832} C_DIS
LIN {X -118.7358,Y 52.0287,Z 159,A 155.2814,B 14.7748,C -0.173,E1 14.6296,E2 294.2705} C_DIS
LIN {X -117.1896,Y 55.4223,Z 159,A 153.6466,B 14.7748,C -0.1779,E1 14.6315,E2 295.9017} C_DIS
LIN {X -115.797,Y 58.2767,Z 159,A 152.2315,B 14.7748,C -0.1815,E1 14.6333,E2 297.3161} C_DIS
LIN {X -114.3367,Y 61.094,Z 159,A 150.9041,B 14.7746,C -0.1873,E1 14.635,E2 298.6333} C_DIS
LIN {X -113.0813,Y 63.3871,Z 159,A 149.6332,B 14.7746,C -0.1873,E1 14.6367,E2 299.9158} C_DIS
LIN {X -111.1887,Y 66.6518,Z 159,A 147.9528,B 14.7746,C -0.1914,E1 14.6391,E2 301.5954} C_DIS
LIN {X -109.2242,Y 69.8238,Z 159,A 146.2066,B 14.7746,C -0.1931,E1 14.6417,E2 303.3506} C_DIS
LIN {X -107.2107,Y 72.878,Z 159,A 144.7123,B 14.7745,C -0.2005,E1 14.644,E2 304.8289} C_DIS
LIN {X -105.3793,Y 75.5016,Z 159,A 143.1285,B 14.7745,C -0.1996,E1 14.6466,E2 306.4302} C_DIS
LIN {X -102.8509,Y 78.9114,Z 159,A 141.2299,B 14.7745,C -0.2036,E1 14.6498,E2 308.329} C_DIS
LIN {X -100.2104,Y 82.2388,Z 159,A 139.3402,B 14.7744,C -0.2078,E1 14.6531,E2 310.2177} C_DIS
LIN {X -97.4487,Y 85.4936,Z 159,A 137.4319,B 14.7744,C -0.2116,E1 14.6565,E2 312.1261} C_DIS
LIN {X -94.6212,Y 88.6128,Z 159,A 135.6097,B 14.7742,C -0.2169,E1 14.66,E2 313.9417} C_DIS
LIN {X -91.6683,Y 91.6645,Z 159,A 133.6548,B 14.7742,C -0.219,E1 14.6638,E2 315.9032} C_DIS
LIN {X -88.601,Y 94.6322,Z 159,A 131.7637,B 14.7742,C -0.2229,E1 14.6676,E2 317.7926} C_DIS
LIN {X -85.4809,Y 97.4597,Z 159,A 129.8839,B 14.7742,C -0.2262,E1 14.6716,E2 319.6723} C_DIS
LIN {X -82.2423,Y 100.2075,Z 159,A 128.0046,B 14.7741,C -0.2299,E1 14.6756,E2 321.5498} C_DIS
LIN {X -79.1222,Y 102.6893,Z 159,A 126.2844,B 14.774,C -0.2345,E1 14.6793,E2 323.2632} C_DIS
LIN {X -76.2597,Y 104.8321,Z 159,A 124.664,B 14.774,C -0.2363,E1 14.683,E2 324.8864} C_DIS
LIN {X -73.3399,Y 106.895,Z 159,A 123.1576,B 14.7739,C -0.2412,E1 14.6864,E2 326.3827} C_DIS
LIN {X -70.6976,Y 108.6607,Z 159,A 121.6441,B 14.7739,C -0.2407,E1 14.69,E2 327.9071} C_DIS
Enddeposition()
END
